# B&R Automation Studio project 8238 (part 23)

#### libTestUse.fun - Exported functions and function blocks
```iecst
(********************************************************************
 * COPYRIGHT -- Herbert Kannegiesser GmbH
 ********************************************************************
 * Library: libTestUse
 * File: libTestUse.fun
 * Author: hunholz
 * Created: March 06, 2012
 ********************************************************************
 * Functions and function blocks of library libTestUse
 ********************************************************************)

FUNCTION_BLOCK TestUser_SetMode (*Versetzt die Anwendung in unterschiedliche Testmodi*)
	VAR_INPUT
		enable : BOOL;
		wMode : UINT;
		pStruc : UDINT;
	END_VAR
	VAR_OUTPUT
		status : UINT;
	END_VAR
	VAR
		_wSetModeState : UINT;
	END_VAR
END_FUNCTION_BLOCK

FUNCTION_BLOCK TestUser_RunTest (*Zyklische Bearbeitung des Tests*)
	VAR_INPUT
		enable : BOOL;
		wMode : UINT;
		pStruc : UDINT;
	END_VAR
	VAR_OUTPUT
		status : UINT;
	END_VAR
	VAR
		_CmdTest : REFERENCE TO TestUser_CmdTest_typ;
		_i : UINT;
		_wCommand : REFERENCE TO UINT;
		_CmdResult : REFERENCE TO ARRAY[0..1] OF UINT;
		_bResult : USINT;
		_wResult : UINT;
		_wXORStatus : UINT;
		_j : UINT;
		_BatchLoad : REFERENCE TO ARRAY[0..3] OF BatchLoad_typ;
		_Batch : REFERENCE TO ARRAY[0..30] OF Batch_typ;
		_BatchUnload : REFERENCE TO ARRAY[0..2] OF Batch_typ;
		_BatchLoadTrig : REFERENCE TO ARRAY[0..3] OF BatchLoadTrig_typ;
		_BatchTrig : REFERENCE TO BatchTrig_typ;
		_BatchUnloadTrig : REFERENCE TO BatchUnloadTrig_typ;
		_xBatchLoadOk : BOOL;
		_xBatchOk : BOOL;
		_xBatchUnloadOk : BOOL;
		_TonShiftClck1 : TON;
		_TonShiftClck2 : TON;
		_wShiftStep : UINT;
		_lBatchNo : UDINT;
		_pBatchNo : REFERENCE TO UDINT;
		_GetTime : DTGetTime;
		_sValue : STRING[10];
		_xBatchForLoadingOk : REFERENCE TO BOOL;
		_enMachineState : REFERENCE TO UDINT;
		_wMachineStateTxt : REFERENCE TO UINT;
		_lMachineStateAtt1 : REFERENCE TO UDINT;
		_lMachineStateAtt2 : REFERENCE TO UDINT;
		_wMachineStateCnt : UINT;
		_Ton1sClck2 : TON;
		_Ton1sClck1 : TON;
	END_VAR
END_FUNCTION_BLOCK

FUNCTION TestUser_StopTask : UINT (*Stoppt Task per Namen*)
	VAR_INPUT
		st_name : UDINT;
	END_VAR
	VAR
		_lTaskIdent : UDINT;
	END_VAR
END_FUNCTION
```

### Program Logical/Standard/Kanlink/KGFrameworkShare/Pkg_mnTestUser/mnTestUser (IEC) - Initialisierung des Test

#### mnTestUserCyclic.st - Cyclic code
```iecst
(********************************************************************
 * COPYRIGHT -- Herbert Kannegiesser GmbH
 ********************************************************************
 * Program: mnTestUser
 * File: mnTestUserCyclic.st
 * Author: hunholz
 * Created: March 07, 2012
 ********************************************************************
 * Implementation of program mnTestUser
 ********************************************************************)

PROGRAM _CYCLIC

(* TODO : Add your code here *)

END_PROGRAM
```

#### mnTestUserInit.st - Initialization code
```iecst
(********************************************************************
 * COPYRIGHT -- Herbert Kannegiesser GmbH
 ********************************************************************
 * Program: mnTestUser
 * File: mnTestUserInit.st
 * Author: hunholz
 * Created: March 07, 2012
 ********************************************************************
 * Implementation of program mnTestUser
 ********************************************************************)

PROGRAM _INIT

	IFmnTest.In.pStrucTest := ADR(_CmdTest);

	_CmdTest.pCmd[1] := ADR(mnMasterCmd.Request.Command);
	_CmdTest.pParamMem[1,1] := ADR(mnMasterCmdAd.SetBatch);
	_CmdTest.pParamSize[1,1] := SIZEOF(mnMasterCmdAd.SetBatch);
	_CmdTest.pCmdResult[1] := ADR(mnMasterCmd.Response);

	_CmdTest.pCmd[2] := ADR(mnLoadCmd.Request.Command);
	_CmdTest.pCmdResult[2] := ADR(mnLoadCmd.Response);

	FOR _i := 0 TO wCountCompMN DO

		_CmdTest.pCmd[3 +_i] := ADR(mnCompCmd[_i].Request.Command);
		_CmdTest.pCmdResult[3 + _i] := ADR(mnCompCmd[_i].Response);

	END_FOR

	_CmdTest.pBatchLoad := ADR(BatchLoad);
	_CmdTest.pBatch := ADR(Batch);
	_CmdTest.pBatchUnload := ADR(BatchUnload);
	_CmdTest.pBatchTrig := ADR(BatchTrig);
	_CmdTest.pBatchLoadTrig := ADR(BatchLoadTrig);
	_CmdTest.pBatchUnloadTrig := ADR(BatchUnloadTrig);

	_CmdTest.pBatchForLoadingOk := ADR(mnMasterStatAd.xBatchTransferDataForLoadingOK);
//
//	_CmdTest.pMachineState := ADR(MachineState.wState);
//	_CmdTest.pMachineStateTxt := ADR(MachineState.wStateTxt);
//	_CmdTest.pMachineStateAtt1 := ADR(MachineState.lStateTxtAtt1);
//	_CmdTest.pMachineStateAtt2 := ADR(MachineState.lStateTxtAtt2);

END_PROGRAM
```

#### mnTestUserExit.st - Exit code
```iecst
(********************************************************************
 * COPYRIGHT -- Herbert Kannegiesser GmbH
 ********************************************************************
 * Program: mnTestUser
 * File: mnTestUserExit.st
 * Author: hunholz
 * Created: March 07, 2012
 ********************************************************************
 * Implementation of program mnTestUser
 ********************************************************************)

PROGRAM _EXIT

(* TODO : Add your code here *)

END_PROGRAM
```

#### mnTestUser.var - Local variables
```iecst
(********************************************************************
 * COPYRIGHT -- Herbert Kannegiesser GmbH
 ********************************************************************
 * Program: mnTestUser
 * File: mnTestUser.var
 * Author: hunholz
 * Created: March 07, 2012
 ********************************************************************
 * Local variables of program mnTestUser
 ********************************************************************)
VAR
	_CmdTest : TestUser_CmdTest_typ;
	_i : UINT;
END_VAR
```

- KanLink Release Notes.docx (binary file, 14716 bytes)
### Package Logical/Standard/Kanlink/CAN - CAN Communication Variables

### CAN.var
```iecst
VAR CONSTANT
	MAX_COMM : USINT := 100;
END_VAR
VAR
	Comm : ARRAY[0..MAX_COMM] OF Comm_typ;
END_VAR
VAR CONSTANT
	COMM_CLEAR : Comm_typ := (0);
END_VAR
```

### CAN.typ
```iecst
TYPE
	WET_CAN : 	STRUCT
		ControlSignals : USINT;
		ControlSignals2 : USINT;
		Category : UINT;
		Customer : UINT;
		Weight : UINT;
	END_STRUCT;
	DRY_CAN : 	STRUCT
		ControlSignals : USINT;
		ControlByte2 : USINT;
		Category : UDINT;
		Weight : UINT;
	END_STRUCT;
	DRY_CAN1 : 	STRUCT
		CustomerCode : UDINT;
		BatchCode : UDINT;
	END_STRUCT;
	DRYCAN_comm_typ : 	STRUCT
		ReadFrame : DRY_CAN;
		WriteFrame : DRY_CAN;
		WriteFrame1 : DRY_CAN1;
		EventRead : BOOL;
		EventWrite : BOOL;
		EventWrite1 : BOOL;
	END_STRUCT;
	Batchpart_typ : 	STRUCT
		Wgt : UINT;
		Customer : UDINT;
	END_STRUCT;
	Comm_typ : 	STRUCT
		BagReady : BOOL;
		Unloading : BOOL;
		DropLoad : BOOL;
		LoadDropped : BOOL;
		Category : UDINT;
		Customer : UDINT;
		BatchID : UDINT;
		Weight : UINT;
		Live : BOOL;
		LiveTime : UINT;
		ReadyToLoad : BOOL;
		Loading : BOOL;
		UnloadFinished : BOOL;
		HaltSys : BOOL;
		Batch_QtyRemaining : UINT;
		LoadRecieved : BOOL;
		Transfer : BOOL;
		Batchpart : ARRAY[0..7]OF Batchpart_typ;
		CategoryStr : STRING[11];
		CustomerStr : STRING[11];
	END_STRUCT;
END_TYPE
```

### Program Logical/Standard/Kanlink/kanlink_map (IEC) - *Custom task to convert Kanlink PLC to eVue Comms

#### Variables.var
```iecst
VAR
	bag_2_wieight : INT;
	doubleDrop : BOOL;
END_VAR
```

#### Cyclic.st
```iecst
PROGRAM _CYCLIC

////SDC1 r43
//Comm[1].Customer	:= wash_com_cust_1;
//Comm[1].Category	:= wash_com_cat_1;
//Comm[1].BatchID		:= DByte_TO_4Byte(ADR(wash_com_batch1_1),ADR(wash_com_batch1_2));
//Comm[1].Weight		:= (wash_com_wt_1 * 10);
//
//Comm[1].BagReady	:= r43.sling_ready;
//r43.open_signal	:= 	Comm[1].DropLoad;
//r43.receive_signal	:= 	Comm[1].LoadDropped;
//IF EDGEPOS(Comm[1].LoadDropped) THEN
//	wash_com_cust_1 := 0;
//	wash_com_cat_1  := 0;
//	wash_com_wt_1  := 0;
//	wash_com_batch1_1 := 0;
//	wash_com_batch1_2 := 0;
//END_IF;
//
////SDC2 r45
//Comm[2].Customer	:= wash_com_cust_2;
//Comm[2].Category	:= wash_com_cat_2;
//Comm[2].BatchID		:= DByte_TO_4Byte(ADR(wash_com_batch1_2),ADR(wash_com_batch2_2));
//Comm[2].Weight		:= (wash_com_wt_2 * 10);
//
//Comm[2].BagReady	:= r45.sling_ready;
//r45.open_signal	:= 	Comm[2].DropLoad;
//r45.receive_signal	:= 	Comm[2].LoadDropped;
//IF EDGEPOS(Comm[2].LoadDropped) THEN
//	wash_com_cust_2 := 0;
//	wash_com_cat_2  := 0;
//	wash_com_wt_2  := 0;
//	wash_com_batch1_2 := 0;
//	wash_com_batch2_2 := 0;
//END_IF;
//
////SDC3 r47
//Comm[3].Customer	:= wash_com_cust_3;
//Comm[3].Category	:= wash_com_cat_3;
//Comm[3].BatchID		:= DByte_TO_4Byte(ADR(wash_com_batch1_3),ADR(wash_com_batch2_3));
//Comm[3].Weight		:= (wash_com_wt_3 * 10);
//
//Comm[3].BagReady	:= r47.sling_ready;
//r47.open_signal	:= 	Comm[3].DropLoad;
//r47.receive_signal	:= 	Comm[3].LoadDropped;
//IF EDGEPOS(Comm[3].LoadDropped) THEN
//	wash_com_cust_3 := 0;
//	wash_com_cat_3  := 0;
//	wash_com_wt_3  := 0;
//	wash_com_batch1_3 := 0;
//	wash_com_batch2_3 := 0;
//END_IF;
//
////CDC8 r110
//Comm[4].Customer	:= wash_com_cust_12;
//Comm[4].Category	:= wash_com_cat_12;
//Comm[4].BatchID		:= DByte_TO_4Byte(ADR(wash_com_batch1_12),ADR(wash_com_batch2_12));
//Comm[4].Weight		:= (wash_com_wt_12 * 10);
//
//Comm[4].BagReady	:= r110.sling_ready;
//r110.open_signal	:= 	Comm[4].DropLoad;
//r110.receive_signal	:= 	Comm[4].LoadDropped;
//IF EDGEPOS(Comm[4].LoadDropped) THEN
//	wash_com_cust_12 := 0;
//	wash_com_cat_12  := 0;
//	wash_com_wt_12  := 0;
//	wash_com_batch1_12 := 0;
//	wash_com_batch2_12 := 0;
//END_IF;
//
////CDC5 r113
//Comm[5].Customer	:= wash_com_cust_13;
//Comm[5].Category	:= wash_com_cat_13;
//Comm[5].BatchID		:= DByte_TO_4Byte(ADR(wash_com_batch1_13),ADR(wash_com_batch2_13));
//Comm[5].Weight		:= (wash_com_wt_13 * 10);
//
//Comm[5].BagReady	:= r113.sling_ready;
//r113.open_signal	:= 	Comm[5].DropLoad;
//r113.receive_signal	:= 	Comm[5].LoadDropped;
//IF EDGEPOS(Comm[5].LoadDropped) THEN
//	wash_com_cust_13 := 0;
//	wash_com_cat_13  := 0;
//	wash_com_wt_13  := 0;
//	wash_com_batch1_13 := 0;
//	wash_com_batch2_13 := 0;
//END_IF;
//
//////CDC6 r68
////Comm[6].Customer	:= wash_com_cust_6;
////Comm[6].Category	:= wash_com_cat_6;
////Comm[6].BatchID		:= DByte_TO_4Byte(ADR(wash_com_batch1_6),ADR(wash_com_batch2_6));
////Comm[6].Weight		:= (wash_com_wt_6 * 10);
////
////Comm[6].BagReady	:= r68.sling_ready;
////r68.open_signal	:= 	Comm[6].DropLoad;
////r68.receive_signal	:= 	Comm[6].LoadDropped;
////IF EDGEPOS(Comm[6].LoadDropped) THEN
////	wash_com_cust_6 := 0;
////	wash_com_cat_6  := 0;
////	wash_com_wt_6  := 0;
////	wash_com_batch1_6 := 0;
////	wash_com_batch2_6 := 0;
////END_IF;
////
//////CDC7 r70
////Comm[7].Customer	:= wash_com_cust_7;
////Comm[7].Category	:= wash_com_cat_7;
////Comm[7].BatchID		:= DByte_TO_4Byte(ADR(wash_com_batch1_7),ADR(wash_com_batch2_7));
////Comm[7].Weight		:= (wash_com_wt_7 * 10);
////
////Comm[7].BagReady	:= r70.sling_ready;
////r70.open_signal	:= 	Comm[7].DropLoad;
////r70.receive_signal	:= 	Comm[7].LoadDropped;
////IF EDGEPOS(Comm[7].LoadDropped) THEN
////	wash_com_cust_7 := 0;
////	wash_com_cat_7  := 0;
////	wash_com_wt_7  := 0;
////	wash_com_batch1_7 := 0;
////	wash_com_batch2_7 := 0;
////END_IF;
////
//////SSL1 r1 - Comm[8]
////
////CSL1 r65
//wash_com_cust_14 	:= UDINT_TO_INT(Comm[14].Customer);
//wash_com_cat_14 		:= UDINT_TO_INT(Comm[14].Category);
//wash_com_wt_14 		:= (Comm[14].Weight/10);
//wash_com_batch1_14	:= Get_Lower2Bytes(Comm[14].BatchID);
//wash_com_batch2_14	:= Get_Higher2Bytes(Comm[14].BatchID);
//
//Comm[14].ReadyToLoad		:= r65.sling_ready;
//r65.xfer_in_progress	:= Comm[14].Unloading;
//
//IF EDGEPOS(r65.fire) THEN
//	wash_com_cust_14 := 0;
//	wash_com_cat_14 := 0;
//	wash_com_wt_14 := 0;
//	wash_com_batch1_14 := 0;
//	wash_com_batch2_14 := 0;
//END_IF;
//
////CSL2 r68
//wash_com_cust_15 	:= UDINT_TO_INT(Comm[15].Customer);
//wash_com_cat_15 	:= UDINT_TO_INT(Comm[15].Category);
//wash_com_wt_15 		:= (Comm[15].Weight/10);
//wash_com_batch1_15	:= Get_Lower2Bytes(Comm[15].BatchID);
//wash_com_batch2_15	:= Get_Higher2Bytes(Comm[15].BatchID);
//
//Comm[15].ReadyToLoad	:= r68.sling_ready;
//r68.xfer_in_progress	:= Comm[15].Unloading;
//
//IF EDGEPOS(r68.fire) THEN
//	wash_com_cust_15 := 0;
//	wash_com_cat_15 := 0;
//	wash_com_wt_15 := 0;
//	wash_com_batch1_15 := 0;
//	wash_com_batch2_15 := 0;
//END_IF;
//
////CSL3 r49
//wash_com_cust_11 	:= UDINT_TO_INT(Comm[11].Customer);
//wash_com_cat_11 	:= UDINT_TO_INT(Comm[11].Category);
//wash_com_wt_11 		:= (Comm[11].Weight/10);
//wash_com_batch1_11	:= Get_Lower2Bytes(Comm[11].BatchID);
//wash_com_batch2_11	:= Get_Higher2Bytes(Comm[11].BatchID);
//
//Comm[11].ReadyToLoad	:= r49.sling_ready;
//r49.xfer_in_progress	:= Comm[11].Unloading;
//
//IF EDGEPOS(r49.fire) THEN
//	wash_com_cust_11 := 0;
//	wash_com_cat_11 := 0;
//	wash_com_wt_11 := 0;
//	wash_com_batch1_11 := 0;
//	wash_com_batch2_11 := 0;
//END_IF;

////CDC2 r70  - DOUBLE DROP>
//Comm[1].Customer	:= wash_com_cust_1;
//Comm[1].Category	:= wash_com_cat_1;
//Comm[1].BatchID		:= DByte_TO_4Byte(ADR(wash_com_batch1_1),ADR(wash_com_batch2_1));
////Comm[1].Weight		:= (wash_com_wt_1 * 10);
//
//bag_4_wieight 		:= WORD_TO_INT(plc_info1);  // 2nd Bag wieght - 1 if the wieght is -0 so we know there is 2 bags.
//doubleDrop			:= (bag_2_wieight > 0);
////Build the batch of 2
//
//IF EDGEPOS(r70.loading_signal) THEN // Decider has ran
//	IF doubleDrop THEN
//		Comm[1].Batch_QtyRemaining := 2;
//	ELSE
//		Comm[1].Batch_QtyRemaining := 1;
//	END_IF;
//END_IF;
//
//IF EDGEPOS(r70.state = 2 ) THEN // Bag arrives in the discharger
//	CASE Comm[1].Batch_QtyRemaining OF
//		1:
//			Comm[1].Batchpart[1].Customer := Comm[1].Customer;
//			Comm[1].Batchpart[1].Wgt := (wash_com_wt_1 * 10);
//			Comm[1].Batchpart[2].Customer := 0;
	//			Comm[1].Batchpart[2].Wgt := 0;
//			Comm[1].Weight := (wash_com_wt_1 *10);
//		2:
//			Comm[1].Batchpart[1].Customer := Comm[1].Customer;
//			Comm[1].Batchpart[1].Wgt := (wash_com_wt_1 * 10);
//			Comm[1].Batchpart[2].Customer := Comm[1].Customer;
//			Comm[1].Batchpart[2].Wgt := (bag_2_wieight * 10);
//			Comm[1].Weight := ((wash_com_wt_1 + bag_2_wieight) *10);
//	END_CASE;
//END_IF;
//
//Comm[1].BagReady	:= r70.sling_ready;
//r70.open_signal	:= 	Comm[1].DropLoad;
//r70.receive_signal	:= 	Comm[1].LoadDropped;
//IF EDGEPOS(Comm[1].LoadDropped) THEN
//	wash_com_cust_1 := 0;
//	wash_com_cat_1  := 0;
//	wash_com_wt_1  := 0;
//	wash_com_batch1_1 := 0;
//	wash_com_batch2_1 := 0;
//	// Count down the loads
//	IF 	Comm[1].Batch_QtyRemaining >= 1 THEN
//		Comm[1].Batch_QtyRemaining := Comm[1].Batch_QtyRemaining - 1;
//	ELSE
//		Comm[1].Batch_QtyRemaining := 0;
//	END_IF;
//END_IF;
//

END_PROGRAM
```

### Package Logical/Robo_Drive_Control - Supertrack Robo Drive Control Package

### Robo_Drive.var - Global variables
```iecst
(********************************************************************
 * COPYRIGHT --
 ********************************************************************
 * Package: FC302
 * File: FC302.var
 * Author: D.Jefferys
 * Created: February 08, 2009
 ********************************************************************
 * Variables of package FC302
 ********************************************************************)
VAR CONSTANT
	AlignReceive : USINT := 1;
	AlignRelease : USINT := 0;
	AlignNone : USINT := 2;
	AlignRest : USINT := 3;
END_VAR
VAR
	StartNode : USINT := 0;
	RB : ARRAY[0..MaxRobo] OF FC302_Drive_Typ := [8(0)];
END_VAR
VAR RETAIN
	RB_Retain : ARRAY[0..MaxRobo] OF FC302_Drive_Retain_Typ;
	RB_Posn : ARRAY[0..MaxRobo] OF FC302_Position_Type;
	RB_Perm : ARRAY[0..MaxRobo] OF FC302_Drive_Permanent_Typ;
END_VAR
VAR
	RB_PosnName : ARRAY[0..MaxRobo] OF RoboPositionNames;
	MonitorIdx : USINT := 0;
END_VAR
```

### Library Logical/Robo_Drive_Control/FC302 (IEC) - FC302 Functions Library

#### FC302.typ - Exported data types
```iecst
(********************************************************************
 * COPYRIGHT --
 ********************************************************************
 * Library: FC302
 * File: FC302.typ
 * Author: D.Jefferys
 * Created: February 12, 2009
 ********************************************************************
 * Data types of library FC302
 ********************************************************************)

TYPE
	RoboPositionNames : 	STRUCT
		Name : ARRAY[0..MaxPositions]OF UINT;
		Extra : ARRAY[0..MaxPositions]OF UINT;
	END_STRUCT;
	FC302_Position_Type : 	STRUCT
		Lift : FC032_Drive_Positions_Type;
		Rotate : FC032_Drive_Positions_Type;
	END_STRUCT;
	FC032_Drive_Positions_Type : 	STRUCT
		RefOffset : DINT;
		MaxSpeed : DINT; (*Max speed in mm/sec*)
		CycleCount : DINT; (*Read only for TrackView display only*)
		PositionNow : DINT;
		OperationMode : DINT; (*0=Normal Sequence 1=Manual Operation*)
		IOStatus : DINT; (*I/O Transmitted to TrackView*)
		Monitor : DINT; (*Monitor Values*)
		SeqStep : DINT; (*Sequence Step*)
		Posn : ARRAY[0..MaxPositions]OF DINT;
	END_STRUCT;
	FC302_Drive_Permanent_Typ : 	STRUCT
		Lift : FC302_LiftPermenant;
		Rotate : FC302_RotatePermenant;
	END_STRUCT;
	FC302_LiftPermenant : 	STRUCT
		CycleCount : DINT;
	END_STRUCT;
	FC302_RotatePermenant : 	STRUCT
		CycleCount : DINT;
	END_STRUCT;
	FC302_Drive_Retain_Typ : 	STRUCT
		Lift : FC302_LiftRemanent;
		Rotate : FC302_RotateRemanent;
	END_STRUCT;
	FC302_Drive_Typ : 	STRUCT
		Lift : FC302_Lift;
		Rotate : FC302_Rotate;
	END_STRUCT;
	FC302_RotateRemanent : 	STRUCT
		PosnRef : DINT;
	END_STRUCT;
	FC302_LiftRemanent : 	STRUCT
		PosnRef : DINT;
	END_STRUCT;
	FC302_Lift : 	STRUCT
		SeqStep : UINT;
		Encoder : DINT; (*Encoder raw value from card*)
		PosnActRaw : UDINT; (*Encoder position actual value always positive*)
		PosnAct : DINT;
		PosnNow : DINT; (*Actual calculated position in 100th of mm*)
		PulsePer10th_mm : REAL;
		DistRemain : DINT;
		mmPerHz : REAL;
		RunHz : UINT; (*Calculated run frequency *)
		StopDist : DINT;
		RunForwards : BOOL;
		RunReverse : BOOL;
		RunFreq : UINT; (*Actual drive running frequency *)
		RampStart : DINT; (*Final Ramp Start (ms)*)
		RampTime : DINT; (*Final Ramp Time (ms)*)
		RampMax : DINT; (*Final Ramp Max Time (ms)*)
		CAN : FC302_CAN_Typ;
		Scan : FC302_CAN_Scan_Typ;
		CTW : FC302_CTW_Typ;
		STW : FC302_STW_Typ;
		SeqIn : FC302_ControlIn; (*Inputs from PLC Sequence*)
		SeqOut : FC302_ControlOut; (*Outputs to PLC Sequence*)
		ParaList : ARRAY[0..59]OF FC302_Parameter_Typ;
		Motor : FC302_Motor_Info;
		ParamWrite : FC302_ParamWrite;
		ParameterCount : UINT;
		ModuleOK : BOOL;
	END_STRUCT;
	FC302_Rotate : 	STRUCT
		SeqStep : UINT;
		Encoder : DINT; (*Encoder raw value from card*)
		PosnActRaw : UDINT; (*Encoder position actual value always positive*)
		PosnAct : DINT;
		PosnNow : DINT; (*Actual calculated position in 100ths of degrees*)
		PulsePer100th_Deg : REAL;
		DistRemain : DINT;
		mmPerHz : REAL;
		RunHz : UINT; (*Calculated run frequency *)
		StopDist : DINT;
		RefOffsetDeg : UINT; (*Degrees from 0 of the reference proximity switch in 100ths 50 = 5000*)
		RunForwards : BOOL;
		RunReverse : BOOL;
		RunFreq : UINT; (*Actual drive running frequency *)
		RampStart : DINT; (*Final Ramp Start (ms)*)
		RampTime : DINT; (*Final Ramp Time (ms)*)
		RampMax : DINT; (*Final Ramp Max Time (ms)*)
		CAN : FC302_CAN_Typ;
		CTW : FC302_CTW_Typ;
		STW : FC302_STW_Typ;
		Scan : FC302_CAN_Scan_Typ;
		SeqIn : FC302_ControlIn; (*Inputs from PLC Sequence*)
		SeqOut : FC302_ControlOut; (*Outputs to PLC Sequence*)
		ParaList : ARRAY[0..59]OF FC302_Parameter_Typ;
		Motor : FC302_Motor_Info;
		ParamWrite : FC302_ParamWrite;
		ParameterCount : UINT;
		ModuleOK : BOOL;
	END_STRUCT;
	FC302_ControlIn : 	STRUCT
		DoRef : BOOL;
		AutoTunePosn : UINT; (*Auto tune position number*)
		AutoTuneReceive : BOOL; (*Auto tune for receive alignment*)
		sDevice : STRING[10]; (*CAN Device eg. "SS1.IF2"*)
		sParTblName : STRING[10]; (*Taskname of parameter table*)
		Node : USINT; (*CAN Node of drive*)
		DisableDrive : BOOL; (*Input - Enable drive to run the motor*)
		I_RefPosn : BOOL; (*Input - PLC Input for reference position*)
		I_ForwardLimitOk : BOOL; (*Input - PLC Input for Top/Clockwise limit *)
		I_ReverseLimitOk : BOOL; (*Input - PLC Input for Bottom/Anti-clockwise limit*)
		I_RailOkRelease : BOOL; (*Input - PLC Input for Rail aligned for bag to leave*)
		I_RailOkReceive : BOOL; (*Input - PLC Input for Rail aligned to Receive a bag*)
		JogForwards : BOOL;
		JogReverse : BOOL;
		EStop : BOOL; (*Input - System emergency stop - will stop drive*)
		PosnReq : DINT; (*Input - Required position in mm 10ths / 100ths Deg *)
		MaxSpeed : DINT; (*Input - Max running speed mm/sec *)
		PowerSave : BOOL; (*Input - Not Busy so save power move slower*)
		RailAlign : USINT; (*Input - Rail Align Requirement*)
		Run : BOOL; (*Input - Run Drive*)
	END_STRUCT;
	FC302_ControlOut : 	STRUCT
		PosnNow : INT; (*Output - Actual Position in mm*)
		PosnOk : BOOL; (*Output - Current position ok for release*)
		DriveDisabled : BOOL; (*Output - Drive acknoledge Enable Movement is off*)
		RefComplete : BOOL; (*Output - Drive is referenced and ready to run*)
		AutoTunePosn : UINT; (*Auto tune position number*)
		Status : UINT; (*Output - Drive sequence status 0 = all ok ready*)
	END_STRUCT;
	FC302_CAN_Scan_Typ : 	STRUCT
		Start : TIME;
		End : TIME;
		LastScan : UINT;
		MinScan : UINT;
		MaxScan : UINT;
		StartTrig : BOOL;
		EndTrig : BOOL;
	END_STRUCT;
	FC302_CAN_Typ : 	STRUCT
		ModuleOk : BOOL; (*Module OK*)
		NodeStatus : UINT; (*Node Status*)
		ControlWord : UINT; (*Control Word*)
		StatusWord : UINT; (*Status Word*)
		TargetVelocity : UINT; (*Target Velocity*)
		ControlEffort : UINT; (*Control Effort*)
	END_STRUCT;
	FC302_Parameter_Typ : 	STRUCT
		index : UINT;
		subindex : USINT;
		datalen : USINT;
		data : UDINT;
	END_STRUCT;
	FC302_ParamWrite : 	STRUCT
		ErrorCount : UINT;
		Index : UINT;
		SubIndex : USINT;
	END_STRUCT;
	FC302_STW_Typ : 	STRUCT  (*Status Word Type*)
		ControlReady : BOOL; (*0 = Off tripped  1 = Controls ready*)
		DriveReady : BOOL; (*0 = Drive not ready 1 = Drive ready*)
		CoastingStop : BOOL; (*0 = Drive has released the motor 1 = Operation enabled*)
		Trip : BOOL; (*0 = No error 1 = Drive Tripped*)
		Error : BOOL; (*0 = No error 1 = Drive has an error but not tripped*)
		NotUsed : BOOL;
		TripLock : BOOL; (*0 = No error 1 = Drive is tripped and locked*)
		Warning : BOOL; (*0 = No error 1 = Drive warning has occured*)
		SpeedReference : BOOL; (*0 = Speed not equal to reference 1 = Speed equals reference*)
		BusOperation : BOOL; (*0 = Local operation no bus control 1 = Bus operation enabled *)
		FreqLimitOk : BOOL; (*0 = Frequency limit reached high or low 1 = Between the limits*)
		DriveOverTemp : BOOL; (*0 = Temperature ok 1 = Drive stopped because of over temperature will resume *)
		DriveVoltageFault : BOOL; (*0 = Voltage ok 1 = Drive DC voltage too high or low*)
		DriveTorqueLimit : BOOL; (*0 = Torque ok 1 = Torque (Current) limit in param 4-18 has been exceded *)
		ThermalTimerLimit : BOOL; (*0 = Timer ok 1 = One of the thermal protection timers has exceeded 100%*)
		InOperation : BOOL; (*0 = Stopped 1 = Drive running greater then 0 Hz*)
	END_STRUCT;
	FC302_Motor_Info : 	STRUCT  (*Current Motor Information *)
		Value : INT;
	END_STRUCT;
	FC302_CTW_Typ : 	STRUCT  (*Control Word Type*)
		ExtRefSelectionLSB : BOOL; (*Used to select between the 4 reference values in parameter 3-10*)
		ExtRefSelectionMSB : BOOL; (*Used to select between the 4 reference values in parameter 3-10*)
		DC_Brake : BOOL; (*0 = DC Brake 1 = Ramp *)
		Coasting : BOOL; (*0 = Coasting 1 = No Coasting, selecting 0 will shut off the output transistors.*)
		QuickStop : BOOL; (*0 = QuickStop 1= Ramp, selecting 0 will use parameter 3-81 quick stop ramp time.*)
		HoldOutputFreq : BOOL; (*0 = Hold 1= Ramp, always use Ramp*)
		RampStopStart : BOOL; (*0 = Ramp stop 1 = Start, Normal stsrt / stop*)
		ResetTrip : BOOL; (*0 = Nothing 1 = Reset Trip*)
		Jog : BOOL; (*0 = Normal 1 = Jog, Jog frequency set by parameter 3-19*)
		RampSelection : BOOL; (*0 = Ramp 1 1 = Ramp 2, Select between ramp 1 and 2 3-40 to 3-47 or 3-50 to 3-57*)
		DataValid : BOOL; (*0 = Not Valid 1 = Data Valid, If not valid then the whole control word is ignored.*)
		Relay01Active : BOOL; (*0 = No function*)
		Relay02Active : BOOL; (*0 = No function*)
		ParaSetUpLSB : BOOL; (*Used to select between the 4 different parameter setups*)
		ParaSetUpMSB : BOOL; (*Used to select between the 4 different parameter setups*)
		Reverse : BOOL; (*0 = No reversing 1 = Reversing*)
	END_STRUCT;
END_TYPE
```

#### FC302.var - Exported constants
```iecst
(********************************************************************
 * COPYRIGHT --
 ********************************************************************
 * Library: FC302
 * File: FC302.var
 * Author: D.Jefferys
 * Created: February 12, 2009
 ********************************************************************
 * Constants of library FC302
 ********************************************************************)
VAR CONSTANT
	posnNameNone : UINT := 0;
	posnNameTop : UINT := 1;
	posnNameTopBagIn : UINT := 2;
	posnNameTopBagOut : UINT := 3;
	posnNameBottom : UINT := 4;
	posnNameBottomBagIn : UINT := 5;
	posnNameBottomBagOut : UINT := 6;
	posnNameMiddle : UINT := 7;
	posnNameMiddleBagIn : UINT := 8;
	posnNameMiddleBagOut : UINT := 9;
	posnNameHighLevel : UINT := 10;
	posnNameHighLevelBagIn : UINT := 11;
	posnNameHighLevelBagOut : UINT := 12;
	posnNameLowLevel : UINT := 13;
	posnNameLowLevelBagIn : UINT := 14;
	posnNameLowLevelBagOut : UINT := 15;
	posnNameMidLevel : UINT := 16;
	posnNameMidLevelBagIn : UINT := 17;
	posnNameMidLevelBagOut : UINT := 18;
	posnNameDocking : UINT := 19;
	posnNameDummy : UINT := 20;
	posnNameLoading : UINT := 21;
	posnNameLine : UINT := 22;
	posnNameParking : UINT := 23;
	posnNameRecirculation : UINT := 24;
	posnNameSafety : UINT := 25;
	posnNameWeighing : UINT := 26;
	posnExtraNone : UINT := 0;
	posnExtraLine1 : UINT := 1;
	posnExtraLine2 : UINT := 2;
	posnExtraLine3 : UINT := 3;
	posnExtraLine4 : UINT := 4;
	posnExtraLine5 : UINT := 5;
	posnExtraLine6 : UINT := 6;
	posnExtraLine7 : UINT := 7;
	posnExtraLine8 : UINT := 8;
	posnExtraLine9 : UINT := 9;
	posnExtraLine10 : UINT := 10;
	posnExtraLine11 : UINT := 11;
	posnExtraLine12 : UINT := 12;
	posnExtraLine13 : UINT := 13;
	posnExtraLine14 : UINT := 14;
	posnExtraLine15 : UINT := 15;
	posnExtraLine16 : UINT := 16;
	posnExtraLine17 : UINT := 17;
	posnExtraLine18 : UINT := 18;
	posnExtraLine19 : UINT := 19;
	posnExtraLine20 : UINT := 20;
	posnExtraLine21 : UINT := 21;
	posnExtraLine22 : UINT := 22;
	posnExtraLine23 : UINT := 23;
	posnExtraLine24 : UINT := 24;
	posnExtraLine25 : UINT := 25;
	posnExtraLine26 : UINT := 26;
	posnExtraLine27 : UINT := 27;
	posnExtraLine28 : UINT := 28;
	posnExtraLine29 : UINT := 29;
	posnExtraSeqHeader1 : UINT := 101;
	posnExtraSeqHeader2 : UINT := 102;
	posnExtraSeqHeader3 : UINT := 103;
	posnExtraSeqHeader4 : UINT := 104;
	posnExtraSeqHeader5 : UINT := 105;
	posnExtraSeqHeader6 : UINT := 106;
	posnExtraSeqHeader7 : UINT := 107;
	posnExtraSeqHeader8 : UINT := 108;
	posnExtraSeqHeader9 : UINT := 109;
	posnExtraSeqHeader10 : UINT := 110;
	posnExtraSeqHeader11 : UINT := 111;
	posnExtraSeqHeader12 : UINT := 112;
	posnExtraSeqHeader13 : UINT := 113;
	posnExtraSeqHeader14 : UINT := 114;
	posnExtraSeqHeader15 : UINT := 115;
	posnExtraSeqHeader16 : UINT := 116;
	posnExtraSeqHeader17 : UINT := 117;
	posnExtraSeqHeader18 : UINT := 118;
	posnExtraSeqHeader19 : UINT := 119;
	posnExtraSeqHeader20 : UINT := 120;
	posnExtraSeqHeader21 : UINT := 121;
	posnExtraSeqHeader22 : UINT := 122;
	posnExtraSeqHeader23 : UINT := 123;
	posnExtraSeqHeader24 : UINT := 124;
	posnExtraSeqHeader25 : UINT := 125;
	posnExtraSeqHeader26 : UINT := 126;
	posnExtraSeqHeader27 : UINT := 127;
	posnExtraSeqHeader28 : UINT := 128;
	posnExtraSeqHeader29 : UINT := 129;
	posnExtraSeqHeader30 : UINT := 130;
	posnExtraSeqHeader31 : UINT := 131;
	posnExtraSeqHeader32 : UINT := 132;
	posnExtraSeqHeader33 : UINT := 133;
	posnExtraSeqHeader34 : UINT := 134;
	posnExtraSeqHeader35 : UINT := 135;
	posnExtraSeqHeader36 : UINT := 136;
	posnExtraSeqHeader37 : UINT := 137;
	posnExtraSeqHeader38 : UINT := 138;
	posnExtraSeqHeader39 : UINT := 139;
	posnExtraSeqHeader40 : UINT := 140;
	posnExtraSeqHeader41 : UINT := 141;
	posnExtraSeqHeader42 : UINT := 142;
	posnExtraSeqHeader43 : UINT := 143;
	posnExtraSeqHeader44 : UINT := 144;
	posnExtraSeqHeader45 : UINT := 145;
	posnExtraSeqHeader46 : UINT := 146;
	posnExtraSeqHeader47 : UINT := 147;
	posnExtraSeqHeader48 : UINT := 148;
	posnExtraSeqHeader49 : UINT := 149;
	MaxRobo : USINT := 7;
	MaxPositions : USINT := 29;
	ModeNothing : UINT := 0;
	ModeReference : UINT := 1;
	ModeManualMove : UINT := 2;
	ModePosnTune : UINT := 3;
	ModeMovePosn : UINT := 4;
	ActionNothing : UINT := 0;
	ActionMoveUp : UINT := 1;
	ActionMoveDown : UINT := 2;
	ActionMoveLeft : UINT := 3;
	ActionMoveRight : UINT := 4;
	FC302_SEQ_OK : USINT := 0;
	FC302_SEQ_Disabled : USINT := 1;
	FC302_SEQ_IndexError : USINT := 2;
	FC302_SEQ_SetCANPreOperational : USINT := 3;
	FC302_SEQ_RestartCANnode : USINT := 4;
	FC302_SEQ_ReadParameterTable : USINT := 5;
	FC302_SEQ_WriteParameters : USINT := 6;
	FC302_SEQ_StoreParameters : USINT := 7;
	FC302_SEQ_CheckParamStored : USINT := 8;
	FC302_SEQ_StartCANnode : USINT := 9;
	FC302_SEQ_WaitDriveOperational : USINT := 10;
	FC302_SEQ_Referencing : USINT := 11;
	FC302_SEQ_MotorWiringFault : USINT := 12;
	FC302_SEQ_RefNotFound : USINT := 13;
	FC302_SEQ_ParameterError : USINT := 14;
	FC302_SEQ_RefSwitchFault : USINT := 15;
	FC302_SEQ_AutoTune : USINT := 16;
	FC302_SEQ_Jog : USINT := 17;
	FC302_SEQ_ReleaseSwitchFault : USINT := 18;
	FC302_SEQ_ReceiveSwitchFault : USINT := 19;
	FC302_SEQ_RailNotAligned : USINT := 20;
	FC302_STW_Trip : USINT := 101;
	FC302_STW_Error : USINT := 102;
	FC302_STW_TripLock : USINT := 103;
	FC302_STW_Warning : USINT := 104;
	FC302_STW_DriveOverTemp : USINT := 105;
	FC302_STW_DriveVoltageFault : USINT := 106;
	FC302_STW_DriveTorqueLimit : USINT := 107;
	FC302_STW_ThermalTimeLimit : USINT := 108;
END_VAR
```

#### FC302.fun - Exported functions and function blocks
```iecst
(********************************************************************
 * COPYRIGHT --
 ********************************************************************
 * Library: FC302
 * File: FC302.fun
 * Author: D.Jefferys
 * Created: February 12, 2009
 ********************************************************************
 * Functions and function blocks of library FC302
 ********************************************************************)

FUNCTION_BLOCK FC302_WriteParam
	VAR_INPUT
		enable : BOOL;
		pDevice : UDINT; (*Add your parameter comment*)
		node : USINT; (*Add your parameter comment*)
		index : UINT; (*Add your parameter comment*)
		subindex : USINT; (*Add your parameter comment*)
		data : UDINT; (*Add your parameter comment*)
		bytelen : USINT; (*Add your parameter comment*)
	END_VAR
	VAR_OUTPUT
		status : UINT; (*Add your parameter comment*)
	END_VAR
	VAR
		CANopenSDOWrite8_0 : CANopenSDOWrite8;
	END_VAR
END_FUNCTION_BLOCK

FUNCTION_BLOCK FC302_ReadSTW (*FC302 Read Status Word*)
	VAR_INPUT
		StatusWord : UINT; (*Add your parameter comment*)
	END_VAR
	VAR_OUTPUT
		STW : FC302_STW_Typ; (*Add your parameter comment*)
	END_VAR
END_FUNCTION_BLOCK

FUNCTION_BLOCK FC302_WriteCTW (*Control Word build*)
	VAR_INPUT
		CTW : FC302_CTW_Typ; (*Add your parameter comment*)
	END_VAR
	VAR_OUTPUT
		ControlWord : UINT; (*Add your parameter comment*)
	END_VAR
	VAR
		LocalControlWord : UINT;
	END_VAR
END_FUNCTION_BLOCK

FUNCTION_BLOCK FC302_ReadParamTbl
	VAR_INPUT
		Enable : BOOL;
		adrTableName : UDINT;
		adrDestTable : UDINT;
		ParamLimit : UINT;
	END_VAR
	VAR_OUTPUT
		ParamCount : UINT;
		Status : UINT;
	END_VAR
	VAR
		DatObjInfo_0 : DatObjInfo;
		DatObjRead_0 : DatObjRead;
	END_VAR
END_FUNCTION_BLOCK

FUNCTION_BLOCK FC302_ReadParam (*Read Parameter from Danfoss FC302*)
	VAR_INPUT
		enable : BOOL; (*Add your parameter comment*)
		pDevice : UDINT; (*Add your parameter comment*)
		node : USINT; (*Add your parameter comment*)
		index : UINT; (*Add your parameter comment*)
		subindex : USINT; (*Add your parameter comment*)
	END_VAR
	VAR_OUTPUT
		data : UDINT; (*Add your parameter comment*)
		status : UINT; (*Add your parameter comment*)
	END_VAR
	VAR
		bytelen : USINT; (*Add your parameter comment*)
		CANopenSDORead8_0 : CANopenSDORead8;
	END_VAR
END_FUNCTION_BLOCK
```

#### FC302_WriteParam.ab - Write Parameter to Danfoss FU302 Drive
```automation-basic
(********************************************************************
 * COPYRIGHT --
 ********************************************************************
 * Program: CAN_Open
 * File: FU302_WriteParam.ab
 * Author: D.Jefferys
 * Created: February 10, 2009
 ********************************************************************
 * Implementation of program CAN_Open
 ********************************************************************)

(*TODO: Add your comment here*)
FUNCTION_BLOCK FC302_WriteParam

	CANopenSDOWrite8_0.enable 	= enable
	CANopenSDOWrite8_0.pDevice 	= pDevice
	CANopenSDOWrite8_0.node 	= node
	CANopenSDOWrite8_0.index 	= $2000 + index
	CANopenSDOWrite8_0.subindex = subindex
	memset(ADR(CANopenSDOWrite8_0.data0),0,8)
	memcpy(ADR(CANopenSDOWrite8_0.data0),ADR(data),4)
	CANopenSDOWrite8_0.datalen 	= bytelen

	CANopenSDOWrite8_0 FUB CANopenSDOWrite8()

	status = CANopenSDOWrite8_0.status

END_FUNCTION_BLOCK
```

#### FC302_ReadSTW.ab - FC302 Read Status Word
```automation-basic
(********************************************************************
 * COPYRIGHT --
 ********************************************************************
 * Program: CAN_Open
 * File: FC302_ReadSTW.ab
 * Author: D.Jefferys
 * Created: February 11, 2009
 ********************************************************************
 * Implementation of program CAN_Open
 ********************************************************************)

(*FC302 Read Status Word*)
FUNCTION_BLOCK FC302_ReadSTW

	STW.ControlReady   		= BIT_TST(StatusWord,0)
	STW.DriveReady			= BIT_TST(StatusWord,1)
	STW.CoastingStop		= BIT_TST(StatusWord,2)
	STW.Trip				= BIT_TST(StatusWord,3)
	STW.Error				= BIT_TST(StatusWord,4)
	STW.NotUsed				= BIT_TST(StatusWord,5)
	STW.TripLock			= BIT_TST(StatusWord,6)
	STW.Warning				= BIT_TST(StatusWord,7)
	STW.SpeedReference		= BIT_TST(StatusWord,8)
	STW.BusOperation		= BIT_TST(StatusWord,9)
	STW.FreqLimitOk			= BIT_TST(StatusWord,10)
	STW.InOperation			= BIT_TST(StatusWord,11)
	STW.DriveOverTemp		= BIT_TST(StatusWord,12)
	STW.DriveVoltageFault	= BIT_TST(StatusWord,13)
	STW.DriveTorqueLimit	= BIT_TST(StatusWord,14)
	STW.ThermalTimerLimit	= BIT_TST(StatusWord,15)

END_FUNCTION_BLOCK
```

#### FC302_WriteCTW.ab - FC302 Write Control Word
```automation-basic
(********************************************************************
 * COPYRIGHT --
 ********************************************************************
 * Library: FC302
 * File: FC302_WriteCTW.ab
 * Author: D.Jefferys
 * Created: February 12, 2009
 ********************************************************************
 * Implementation of library FC302
 ********************************************************************)

(*Control Word build*)
FUNCTION_BLOCK FC302_WriteCTW

	LocalControlWord = 0

	IF CTW.ExtRefSelectionLSB THEN
		LocalControlWord = LocalControlWord + 1
	ENDIF
	IF CTW.ExtRefSelectionMSB THEN
		LocalControlWord = LocalControlWord + 2
	ENDIF
	IF CTW.DC_Brake THEN
		LocalControlWord = LocalControlWord + 4
	ENDIF
	IF CTW.Coasting THEN
		LocalControlWord = LocalControlWord + 8
	ENDIF
	IF CTW.QuickStop THEN
		LocalControlWord = LocalControlWord + 16
	ENDIF
	IF CTW.HoldOutputFreq THEN
		LocalControlWord = LocalControlWord + 32
	ENDIF
	IF CTW.RampStopStart THEN
		LocalControlWord = LocalControlWord + 64
	ENDIF
	IF CTW.ResetTrip THEN
		LocalControlWord = LocalControlWord + 128
	ENDIF
	IF CTW.Jog THEN
		LocalControlWord = LocalControlWord + 256
	ENDIF
	IF CTW.RampSelection THEN
		LocalControlWord = LocalControlWord + 512
	ENDIF
	IF CTW.DataValid THEN
		LocalControlWord = LocalControlWord + 1024
	ENDIF
	IF CTW.Relay01Active THEN
		LocalControlWord = LocalControlWord + 2048
	ENDIF
	IF CTW.Relay02Active THEN
		LocalControlWord = LocalControlWord + 4096
	ENDIF
	IF CTW.ParaSetUpLSB THEN
		LocalControlWord = LocalControlWord + 8192
	ENDIF
	IF CTW.ParaSetUpMSB THEN
		LocalControlWord = LocalControlWord + 16384
	ENDIF
	IF CTW.Reverse THEN
		LocalControlWord = LocalControlWord + 32768
	ENDIF

	ControlWord = LocalControlWord

END_FUNCTION_BLOCK
```

#### FC302_ReadParamTbl.ab - Read from a parameter table
```automation-basic
(********************************************************************
 * COPYRIGHT --
 ********************************************************************
 * Library: FC302
 * File: ReadParamTbl.ab
 * Author: D.Jefferys
 * Created: February 13, 2009
 ********************************************************************
 * Implementation of library FC302
 ********************************************************************)

(*Read from a parameter table*)
FUNCTION_BLOCK FC302_ReadParamTbl

	IF Enable THEN

		Status 		= $FFFF ;Set to busy
		ParamCount 	= 0

		DatObjInfo_0.enable = TRUE
		DatObjInfo_0.pName = adrTableName
		DatObjInfo_0 FUB DatObjInfo()

		IF (DatObjInfo_0.status = 0) THEN

			ParamCount 	= UINT(DatObjInfo_0.len / 8)

			IF (ParamCount <= ParamLimit) THEN

				DatObjRead_0.enable 		= TRUE
				DatObjRead_0.ident 			= DatObjInfo_0.ident
				DatObjRead_0.Offset 		= 0
				DatObjRead_0.pDestination 	= adrDestTable
				DatObjRead_0.len 			= DatObjInfo_0.len
				DatObjRead_0 FUB DatObjRead()

				IF DatObjRead_0.status = 0 THEN
					Status = 0 ;Set status to finished
				ENDIF

			ELSE
				Status = 1 ;Too may parameters
			ENDIF

		ENDIF

	ENDIF

END_FUNCTION_BLOCK
```

#### FC302_ReadParam.ab - Read Parameter from Danfoss FC302
```automation-basic
(********************************************************************
 * COPYRIGHT --
 ********************************************************************
 * Library: FC302
 * File: FC302_ReadParam.ab
 * Author: D.Jefferys
 * Created: February 13, 2009
 ********************************************************************
 * Implementation of library FC302
 ********************************************************************)

(*Read Parameter from Danfoss FC302*)
FUNCTION_BLOCK FC302_ReadParam

	status = 65535 ;Busy

	CANopenSDORead8_0.enable 	= enable
	CANopenSDORead8_0.pDevice 	= pDevice
	CANopenSDORead8_0.node 		= node
	CANopenSDORead8_0.index 	= $2000 + index
	CANopenSDORead8_0.subindex 	= subindex

	CANopenSDORead8_0 FUB CANopenSDORead8()

	IF (CANopenSDORead8_0.status = 0) THEN
		data = 0
		memcpy(ADR(data),ADR(CANopenSDORead8_0.data0),CANopenSDORead8_0.datalen)
		status = CANopenSDORead8_0.status
	ENDIF

END_FUNCTION_BLOCK
```

### Data object Logical/Robo_Drive_Control/Param_3kw (Simple, version 4.00.0) - Parameters 3kW Star from Expo

#### Param_3kw.dat
```
(********************************************************************
 * COPYRIGHT --
 ********************************************************************
 * Data object: Param_2kwStar
 * File: Param_2kwStar.dat
 * Author:  D.Jefferys
 * Created: February 12, 2009
 ********************************************************************
 * Data object file: Param_2kwStar.dat
 ********************************************************************)

;Version 4.01 18/12/2012 T.R. Created 3kw instance based on 2.2kw version 4.00
;CAN Module Switch Settings
;--------------------------

;Baudrate
;8 on  7 on  Par 10-01
;8 on  7 off 500kbps
;8 off 7 on  250kbps
;8 off 7 off 125kbps

;Node Number Binary
;1 = 1s
;2 = 2s
;3 = 4s
;4 = 8s
;5 = 16s
;6 = 32s

;
;	!!! DO NOT CHANGE THE SEQUENCE OF THE PARAMETERS
;
; FU parameter to the Ubertragung (only parameter, which deviates from the default values)
;
; 3 kW Star
;
; Index, Subindex, Datatype (Bytes), Setting (DINT) ; Comments
0002,00,01,00000001	; [000] 00-02, Motor Speed 0 - RPM, 1 - Hz
0001,00,01,00000000	; [001] 00-01, Language 0 - English, 1 - German
0011,00,01,00000001	; [002] 00-11, Edit Setup 1
0190,00,01,00000002	; [003] 01-90, Motor Thermal Protection, 2 - Thermistor
0040,00,01,00000000 ; [004] 00-40, Hand On Key on LCP 0 - Disabled No Function
0381,00,04,00000020 ; [005] 03-81, QuickStop ramp time 100 - 1s
0458,00,01,00000001	; [006] 04-58, Missing motor phase function, 1 - Trip 100ms
0854,00,01,00000001	; [007] 08-54, Reversing select 1 - Bus only 3 - Bus and Terminal
0211,00,02,00000300	; [008] 02-11, Brake resistor 100 Ohm
0212,00,04,00001500	; [009] 02-12, Brake power limit 200 Watt
0213,00,01,00000002	; [010] 02-13, Brake check 2 - Alarm
1426,00,01,00000000 ; [011] 14-26, Trip delay at inverter fault 0 = Disabled
0803,00,04,00000002 ; [012] 08-03, Control Word Timeout Time 10 = 1Sec
0804,00,01,00000002	; [013] 08-04, Control Word Timeout Function 2 - Stop with auto restart
0801,00,01,00000000	; [014] 08-01, Control Site, 0 - Controlword & digital only
0223,00,01,00000005	; [015] 02-23, Active brake delay 0,3 s
1761,00,01,00000002	; [016] 17-61, Encoder Signal Monitoring (Encoder faulty), 2 - Trip
1710,00,01,00000001	; [017] 17-10, Encoder Signal Type 1 - TTL
1711,00,02,00001024	; [018] 17-11, Encoder Resolution 1024 Pulse
0430,00,01,00000001 ; [019] 04-30, Motor Feedback Loss Function, 1 - Warning, 2* - Trip
0431,00,02,00000300 ; [020] 04-31, Motor Feedback Speed Error RPM, 0-600, 300*
0226,00,02,00005000	; [021] 02-26, Torque Ref, 50,00%
0228,00,02,00000200	; [022] 02-28, Gain Boost Factor, 2,00% 0-4% ***************************
0519,00,01,00000003	; [023] 05-19, Terminal 37 Safe Stop, 3 - Safe Stop Warning
0120,00,04,00000300	; [024] 01-20, Motor Power 3kW
0101,00,01,00000003	; [025] 01-01, Motor Control Principle, 3 - Flux with motor feedback
0122,00,02,00000400	; [026] 01-22, Motor voltage 400 V
0123,00,02,00000050	; [027] 01-23, Motor frequency 50 Hz
0162,00,02,00000100	; [028] 01-62, Slip compenstation 100%
0410,00,01,00000002	; [029] 04-10, Motor speed direction, 2 - both directions
0540,00,01,00000032	; [030] 05-40, [0] Relay 1 Function, 32 - Mech brake ctrl
0540,01,01,00000032	; [031] 05-40, [1] Relay 2 Function, 32 - Mech brake ctrl
0802,00,01,00000003 ; [032] 08-02, Control Site 3 - Option A CAN Bus
0102,00,01,00000002	; [033] 01-02, Flux Motor Feeback Source 2 - MCB102
0125,00,02,00001420	; [034] 01-25, Motor nominal speed 1420 rpm
0702,00,02,00000070	; [035] 07-02, Speed PID proportionl gain 0,070
0700,00,01,00000002	; [036] 07-00, Speed PID Feedback Source 2 - MCB102
0172,00,01,00000006	; [037] 01-72, Start function, 6 - Hoist Mech. Brake Rel
0210,00,01,00000001	; [038] 02-10, Brake Function, 1 - Resistor brake
1410,00,01,00000005	; [039] 14-10, Mains failure, 3 - Coasting 5 - Kenetic backup , trip
0193,00,01,00000006	; [040] 01-93, Thermistor source, 6 - Digital Input 33
0100,00,01,00000001	; [041] 01-00, Configuration mode, 1 - Closed loop with encoder
0139,00,01,00000004	; [042] 01-39, Motor poles, 4
0511,00,01,00000000	; [043] 05-11, Terminal 19, 0 - No Operation
0512,00,01,00000000	; [044] 05-12, Terminal 27, 0 - No Operation
0513,00,01,00000000	; [045] 05-13, Terminal 29, 0 - No Operation
0514,00,01,00000004	; [046] 05-14, Terminal 32, 4 - Quick Stop
0510,00,01,00000000	; [047] 05-10, Terminal 18, 0 - No Operation
0175,00,02,00000015	; [048] 01-75, Start Speed, 1,5 Hz
0222,00,02,00000005	; [049] 02-22, Activate Brake Speed ?en bei 0,5 Hz
0124,00,04,00000750	; [050] 01-24, Motor current 7.5 A
0341,00,04,00000100	; [051] 03-41, Ramp 1 ramp up time (1 Sec to 50 Hz)
0342,00,04,00000100	; [052] 03-42, Ramp 1 ramp down time (1 Sec to  0 Hz)
0414,00,02,00001000	; [053] 04-14, Motor Speed High Limit 100,0 Hz
0220,00,04,00000260	; [054] 02-20, Release brake current 2,6 A
(*0130,00,04,00029763	; [---] 01-30, Stator resistance (Rs) 2,9763 Ohm
0131,00,04,00022212	; [---] 01-31, Rotor resistance (Rr) 2,2212 Ohm*)
(*0134,00,04,00031036	; [---] 01-34, Rotor leakage reactance (X2) 3,1036 Ohm*)
;0136,00,04,01803904	; [---] 01-36, Iron loss resistance (Rfe) 1803,904 Ohm
;0135,00,04,00653996	; [---] 01-35, Main reactance (Xh) 65,3996 Ohm
0416,00,02,00002500	; [055] 04-16, Torque limit motor mode, 160,0 - % NOW 250%
0417,00,02,00001600	; [056] 04-17, Torque limit generator mode, 160,0 %
;0133,00,04,00031036	; [---] 01-33, Stator leakage reactance (X1), 3,1036 Ohm
0303,00,04,00100000	; [057] 03-03, Maximum Reference, 100,000
0418,00,04,00002100	; [058] 04-18, Current Limit 172,0 % - NOW 210%
0851,00,01,00000003	; [0] 08-51, Quick stop Logical OR
```

### Data object Logical/Robo_Drive_Control/Param_2_2kwStar (Simple, version 4.00.0) - Parameters 2.2kW Star

#### Param_2_2kwStar.dat
```
(********************************************************************
 * COPYRIGHT --
 ********************************************************************
 * Data object: Param_2kwStar
 * File: Param_2kwStar.dat
 * Author:  D.Jefferys
 * Created: February 12, 2009
 ********************************************************************
 * Data object file: Param_2kwStar.dat
 ********************************************************************)

;Version 2.00 18/10/2010 D.J. Added 14-26 Trip Delay - Disabled, Changed 14-10 from 3 (Coasting) to 5 (Kenetic Backup + Trip)
;Version 3.00 03/11/2010 D.J. Added CAN Switch Settings
;Version 4.00 02/11/2011 D.J. Added Parameter 40 - Hand on Key on LCP now Disabled

;CAN Module Switch Settings
;--------------------------

;Baudrate
;8 on  7 on  Par 10-01
;8 on  7 off 500kbps
;8 off 7 on  250kbps
;8 off 7 off 125kbps

;Node Number Binary
;1 = 1s
;2 = 2s
;3 = 4s
;4 = 8s
;5 = 16s
;6 = 32s

;
;	!!! DO NOT CHANGE THE SEQUENCE OF THE PARAMETERS
;
; FU parameter to the Ubertragung (only parameter, which deviates from the default values)
;
; 2.2 kW Star
;
; Index, Subindex, Datatype (Bytes), Setting (DINT) ; Comments
0002,00,01,00000001	; [000] 00-02, Motor Speed 0 - RPM, 1 - Hz
0001,00,01,00000000	; [001] 00-01, Language 0 - English, 1 - German
0011,00,01,00000001	; [002] 00-11, Edit Setup 1
0190,00,01,00000002	; [003] 01-90, Motor Thermal Protection, 2 - Thermistor
0040,00,01,00000000 ; [---] 00-40, Hand On Key on LCP 0 - Disabled No Function
0381,00,04,00000050 ; [000] 03-81, QuickStop ramp time 100 - 1s
0458,00,01,00000001	; [004] 04-58, Missing motor phase function, 1 - Trip 100ms
0854,00,01,00000001	; [005] 08-54, Reversing select 1 - Bus only 3 - Bus and Terminal
0211,00,02,00000120	; [006] 02-11, Brake resistor 120 Ohm
0212,00,04,00001200	; [007] 02-12, Brake power limit 1200 Watt
0213,00,01,00000002	; [008] 02-13, Brake check 2 - Alarm
1426,00,01,00000000 ; [---] 14-26, Trip delay at inverter fault 0 = Disabled
0803,00,04,00000002 ; [000] 08-03, Control Word Timeout Time 10 = 1Sec
0804,00,01,00000002	; [009] 08-04, Control Word Timeout Function 2 - Stop with auto restart
0801,00,01,00000002	; [010] 08-01, Control Site, 2 - Controlword only
0223,00,01,00000005	; [011] 02-23, Active brake delay 0,3 s
1761,00,01,00000002	; [012] 17-61, Encoder Signal Monitoring (Encoder faulty), 2 - Trip
1710,00,01,00000001	; [013] 17-10, Encoder Signal Type 1 - TTL
1711,00,02,00001024	; [014] 17-11, Encoder Resolution 1024 Pulse
0430,00,01,00000001 ; [015] 04-30, Motor Feedback Loss Function, 1 - Warning, 2* - Trip
0431,00,02,00000300 ; [016] 04-31, Motor Feedback Speed Error RPM, 0-600, 300*
0226,00,02,00005000	; [015] 02-26, Torque Ref, 50,00%
0228,00,02,00000200	; [016] 02-28, Gain Boost Factor, 2,00% 0-4% ***************************
0519,00,01,00000003	; [017] 05-19, Terminal 37 Safe Stop, 3 - Safe Stop Warning
0120,00,04,00000220	; [018] 01-20, Motor Power 2.2kW
0101,00,01,00000003	; [019] 01-01, Motor Control Principle, 3 - Flux with motor feedback
0122,00,02,00000400	; [020] 01-22, Motor voltage 400 V
0123,00,02,00000050	; [021] 01-23, Motor frequency 50 Hz
0162,00,02,00000100	; [022] 01-62, Slip compenstation 100%
0410,00,01,00000002	; [023] 04-10, Motor speed direction, 2 - both directions
0540,00,01,00000032	; [024] 05-40, [0] Relay 1 Function, 32 - Mech brake ctrl
0540,01,01,00000032	; [025] 05-40, [1] Relay 2 Function, 32 - Mech brake ctrl
0802,00,01,00000003 ; [---] 08-02, Control Site 3 - Option A CAN Bus
0102,00,01,00000002	; [026] 01-02, Flux Motor Feeback Source 2 - MCB102
0125,00,02,00001400	; [027] 01-25, Motor nominal speed 1440 rpm
0702,00,02,00000070	; [028] 07-02, Speed PID proportionl gain 0,070
0700,00,01,00000002	; [029] 07-00, Speed PID Feedback Source 2 - MCB102
0172,00,01,00000006	; [030] 01-72, Start function, 6 - Hoist Mech. Brake Rel
0210,00,01,00000001	; [031] 02-10, Brake Function, 1 - Resistor brake
1410,00,01,00000005	; [032] 14-10, Mains failure, 3 - Coasting 5 - Kenetic backup , trip
0193,00,01,00000006	; [033] 01-93, Thermistor source, 6 - Digital Input 33
0100,00,01,00000001	; [034] 01-00, Configuration mode, 1 - Closed loop with encoder
0139,00,01,00000004	; [035] 01-39, Motor poles, 4
0511,00,01,00000000	; [036] 05-11, Terminal 19, 0 - No Operation
0512,00,01,00000000	; [037] 05-12, Terminal 27, 0 - No Operation
0513,00,01,00000000	; [038] 05-13, Terminal 29, 0 - No Operation
0510,00,01,00000000	; [039] 05-10, Terminal 18, 0 - No Operation
0175,00,02,00000015	; [040] 01-75, Start Speed, 1,5 Hz
0222,00,02,00000005	; [041] 02-22, Activate Brake Speed ?en bei 0,5 Hz
0124,00,04,00000520	; [042] 01-24, Motor current 5,2 A
0341,00,04,00000100	; [043] 03-41, Ramp 1 ramp up time (1 Sec to 50 Hz)
0342,00,04,00000100	; [044] 03-42, Ramp 1 ramp down time (1 Sec to  0 Hz)
0414,00,02,00001000	; [045] 04-14, Motor Speed High Limit 100,0 Hz
0220,00,04,00000260	; [046] 02-20, Release brake current 2,6 A
0130,00,04,00029763	; [047] 01-30, Stator resistance (Rs) 2,9763 Ohm
0131,00,04,00022212	; [048] 01-31, Rotor resistance (Rr) 2,2212 Ohm
0134,00,04,00031036	; [049] 01-34, Rotor leakage reactance (X2) 3,1036 Ohm
;0136,00,04,01803904	; [050] 01-36, Iron loss resistance (Rfe) 1803,904 Ohm
;0135,00,04,00653996	; [051] 01-35, Main reactance (Xh) 65,3996 Ohm
0416,00,02,00002500	; [052] 04-16, Torque limit motor mode, 160,0 - % NOW 250%
0417,00,02,00001600	; [053] 04-17, Torque limit generator mode, 160,0 %
;0133,00,04,00031036	; [054] 01-33, Stator leakage reactance (X1), 3,1036 Ohm
0303,00,04,00100000	; [055] 03-03, Maximum Reference, 100,000
0418,00,04,00002500	; [056] 04-18, Current Limit 172,0 % - NOW 250%
```

### Data object Logical/Robo_Drive_Control/ParamD15 (Simple, version 4.00.0) - Parameters 1.5kW Star Disable Drive feedback

#### ParamD15.dat
```
(********************************************************************
 * COPYRIGHT --
 ********************************************************************
 * Data object: Param_1_5kwStar
 * File: Param_1_5kwStar.dat
 * Author:  D.Jefferys
 * Created: October 2, 2009
 ********************************************************************
 * Data object file: Param_1_5kwStar.dat
 ********************************************************************)

;Version 2.00 18/10/2010 D.J. Added 14-26 Trip Delay - Disabled, Changed 14-10 from 3 (Coasting) to 5 (Kenetic Backup + Trip)
;Version 3.00 03/11/2010 D.J. Added CAN Switch Settings
;Version 4.00 02/11/2011 D.J. Added Parameter 40 - Hand on Key on LCP now Disabled

;CAN Module Switch Settings
;--------------------------

;Baudrate
;8 on  7 on  Par 10-01
;8 on  7 off 500kbps
;8 off 7 on  250kbps
;8 off 7 off 125kbps

;Node Number Binary
;1 = 1s
;2 = 2s
;3 = 4s
;4 = 8s
;5 = 16s
;6 = 32s

;
;	!!! DO NOT CHANGE THE SEQUENCE OF THE PARAMETERS
;
; FU parameter to the Ubertragung (only parameter, which deviates from the default values)
;
; 1.5 kW Star
;
; Index, Subindex, Datatype (Bytes), Setting (DINT) ; Comments
0002,00,01,00000001	; [000] 00-02, Motor Speed 0 - RPM, 1 - Hz
0001,00,01,00000000	; [001] 00-01, Language 0 - English, 1 - German
0011,00,01,00000001	; [002] 00-11, Edit Setup 1
0190,00,01,00000000	; [003] 01-90, Motor Thermal Protection, 2 - Thermistor
0040,00,01,00000000 ; [---] 00-40, Hand On Key on LCP 0 - Disabled No Function
0381,00,04,00000050 ; [000] 03-81, QuickStop ramp time 100 - 1s
0458,00,01,00000001	; [004] 04-58, Missing motor phase function, 1 - Trip 100ms
0854,00,01,00000001	; [005] 08-54, Reversing select 1 - Bus only 3 - Bus and Terminal
0211,00,02,00000310	; [006] 02-11, Brake resistor 120 Ohm
0212,00,04,00001200	; [007] 02-12, Brake power limit 1200 Watt
0213,00,01,00000002	; [008] 02-13, Brake check 2 - Alarm
1426,00,01,00000000 ; [---] 14-26, Trip delay at inverter fault 0 = Disabled
0803,00,04,00000002 ; [000] 08-03, Control Word Timeout Time 10 = 1Sec
0804,00,01,00000002	; [009] 08-04, Control Word Timeout Function 2 - Stop with auto restart
0801,00,01,00000002	; [010] 08-01, Control Site, 2 - Controlword only
0223,00,01,00000005	; [011] 02-23, Active brake delay 0,3 s
1761,00,01,00000000	;********************** [012] 17-61, Encoder Signal Monitoring (Encoder faulty), 2 - Trip Changed for testing.
1710,00,01,00000001	; [013] 17-10, Encoder Signal Type 1 - TTL
1711,00,02,00001024	; [014] 17-11, Encoder Resolution 1024 Pulse
0430,00,01,00000001 ; [015] 04-30, Motor Feedback Loss Function, 1 - Warning, 2* - Trip
0431,00,02,00000300 ; [016] 04-31, Motor Feedback Speed Error RPM, 0-600, 300*
0226,00,02,00005000	; [015] 02-26, Torque Ref, 50,00%
0228,00,02,00000200	; [016] 02-28, Gain Boost Factor, 2,00% 0-4% ***************************
0519,00,01,00000003	; [017] 05-19, Terminal 37 Safe Stop, 3 - Safe Stop Warning
0120,00,04,00000150	; [018] 01-20, Motor Power 1.5kW
0101,00,01,00000003	; [019] 01-01, Motor Control Principle, 3 - Flux with motor feedback
0122,00,02,00000400	; [020] 01-22, Motor voltage 400 V
0123,00,02,00000050	; [021] 01-23, Motor frequency 50 Hz
0162,00,02,00000100	; [022] 01-62, Slip compenstation 100%
0410,00,01,00000002	; [023] 04-10, Motor speed direction, 2 - both directions
0540,00,01,00000032	; [024] 05-40, [0] Relay 1 Function, 32 - Mech brake ctrl
0540,01,01,00000032	; [025] 05-40, [1] Relay 2 Function, 32 - Mech brake ctrl
0802,00,01,00000003 ; [---] 08-02, Control Site 3 - Option A CAN Bus
0102,00,01,00000002	; [026] 01-02, Flux Motor Feeback Source 2 - MCB102
0125,00,02,00001400	; [027] 01-25, Motor nominal speed 1440 rpm
0702,00,02,00000070	; [028] 07-02, Speed PID proportionl gain 0,070
0700,00,01,00000002	; [029] 07-00, Speed PID Feedback Source 2 - MCB102
0172,00,01,00000006	; [030] 01-72, Start function, 6 - Hoist Mech. Brake Rel
0210,00,01,00000001	; [031] 02-10, Brake Function, 1 - Resistor brake
1410,00,01,00000005	; [032] 14-10, Mains failure, 3 - Coasting 5 - Kenetic backup , trip
0193,00,01,00000006	; [033] 01-93, Thermistor source, 6 - Digital Input 33
0100,00,01,00000001	; [034] 01-00, Configuration mode, 1 - Closed loop with encoder
0139,00,01,00000004	; [035] 01-39, Motor poles, 4
0511,00,01,00000000	; [036] 05-11, Terminal 19, 0 - No Operation
0512,00,01,00000000	; [037] 05-12, Terminal 27, 0 - No Operation
0513,00,01,00000000	; [038] 05-13, Terminal 29, 0 - No Operation
0510,00,01,00000000	; [039] 05-10, Terminal 18, 0 - No Operation
0175,00,02,00000015	; [040] 01-75, Start Speed, 1,5 Hz
0222,00,02,00000005	; [041] 02-22, Activate Brake Speed ?en bei 0,5 Hz
0124,00,04,00000360	; [042] 01-24, Motor current 5,2 A
0341,00,04,00000100	; [043] 03-41, Ramp 1 ramp up time (1 Sec to 50 Hz)
0342,00,04,00000100	; [044] 03-42, Ramp 1 ramp down time (1 Sec to  0 Hz)
0414,00,02,00001000	; [045] 04-14, Motor Speed High Limit 100,0 Hz
0220,00,04,00000180	; [046] 02-20, Release brake current 1,8 A - About Half of motor A?
;0130,00,04,00029763	; [047] 01-30, Stator resistance (Rs) 2,9763 Ohm
;0131,00,04,00022212	; [048] 01-31, Rotor resistance (Rr) 2,2212 Ohm
;0134,00,04,00031036	; [049] 01-34, Rotor leakage reactance (X2) 3,1036 Ohm
;0136,00,04,01803904	; [050] 01-36, Iron loss resistance (Rfe) 1803,904 Ohm
;0135,00,04,00653996	; [051] 01-35, Main reactance (Xh) 65,3996 Ohm
0416,00,02,00002500	; [052] 04-16, Torque limit motor mode, 160,0 - % NOW 250%
0417,00,02,00001600	; [053] 04-17, Torque limit generator mode, 160,0 %
;0133,00,04,00031036	; [054] 01-33, Stator leakage reactance (X1), 3,1036 Ohm
0303,00,04,00100000	; [055] 03-03, Maximum Reference, 100,000
0418,00,04,00001720	; [056] 04-18, Current Limit 172,0 % - NOW 250%
```

### Data object Logical/Robo_Drive_Control/Param_1_5kwStar_expo (Simple, version 4.00.0) - Parameters 1.5kW Star

#### Param_1_5kwStar.dat
```
(********************************************************************
 * COPYRIGHT --
 ********************************************************************
 * Data object: Param_1_5kwStar
 * File: Param_1_5kwStar.dat
 * Author:  D.Jefferys
 * Created: October 2, 2009
 ********************************************************************
 * Data object file: Param_1_5kwStar.dat
 ********************************************************************)

;Version 2.00 18/10/2010 D.J. Added 14-26 Trip Delay - Disabled, Changed 14-10 from 3 (Coasting) to 5 (Kenetic Backup + Trip)
;Version 3.00 03/11/2010 D.J. Added CAN Switch Settings
;Version 4.00 02/11/2011 D.J. Added Parameter 40 - Hand on Key on LCP now Disabled

;CAN Module Switch Settings
;--------------------------

;Baudrate
;8 on  7 on  Par 10-01
;8 on  7 off 500kbps
;8 off 7 on  250kbps
;8 off 7 off 125kbps

;Node Number Binary
;1 = 1s
;2 = 2s
;3 = 4s
;4 = 8s
;5 = 16s
;6 = 32s

;
;	!!! DO NOT CHANGE THE SEQUENCE OF THE PARAMETERS
;
; FU parameter to the Ubertragung (only parameter, which deviates from the default values)
;
; 1.5 kW Star
;
; Index, Subindex, Datatype (Bytes), Setting (DINT) ; Comments
0002,00,01,00000001	; [000] 00-02, Motor Speed 0 - RPM, 1 - Hz
0001,00,01,00000000	; [001] 00-01, Language 0 - English, 1 - German
0011,00,01,00000001	; [002] 00-11, Edit Setup 1
0190,00,01,00000000	; [003] 01-90, Motor Thermal Protection, 2 - Thermistor
0040,00,01,00000000 ; [---] 00-40, Hand On Key on LCP 0 - Disabled No Function
0381,00,04,00000050 ; [000] 03-81, QuickStop ramp time 100 - 1s
0458,00,01,00000001	; [004] 04-58, Missing motor phase function, 1 - Trip 100ms
0854,00,01,00000001	; [005] 08-54, Reversing select 1 - Bus only 3 - Bus and Terminal
0211,00,02,00000310	; [006] 02-11, Brake resistor 120 Ohm
0212,00,04,00001200	; [007] 02-12, Brake power limit 1200 Watt
0213,00,01,00000002	; [008] 02-13, Brake check 2 - Alarm
1426,00,01,00000000 ; [---] 14-26, Trip delay at inverter fault 0 = Disabled
0803,00,04,00000002 ; [000] 08-03, Control Word Timeout Time 10 = 1Sec
0804,00,01,00000002	; [009] 08-04, Control Word Timeout Function 2 - Stop with auto restart
0801,00,01,00000002	; [010] 08-01, Control Site, 2 - Controlword only
0223,00,01,00000005	; [011] 02-23, Active brake delay 0,3 s
1761,00,01,00000002	; [012] 17-61, Encoder Signal Monitoring (Encoder faulty), 2 - Trip Changed for testing.
1710,00,01,00000001	; [013] 17-10, Encoder Signal Type 1 - TTL
1711,00,02,00001024	; [014] 17-11, Encoder Resolution 1024 Pulse
0430,00,01,00000001 ; [015] 04-30, Motor Feedback Loss Function, 1 - Warning, 2* - Trip
0431,00,02,00000300 ; [016] 04-31, Motor Feedback Speed Error RPM, 0-600, 300*
0226,00,02,00005000	; [015] 02-26, Torque Ref, 50,00%
0228,00,02,00000200	; [016] 02-28, Gain Boost Factor, 2,00% 0-4% ***************************
0519,00,01,00000003	; [017] 05-19, Terminal 37 Safe Stop, 3 - Safe Stop Warning
0120,00,04,00000150	; [018] 01-20, Motor Power 1.5kW
0101,00,01,00000003	; [019] 01-01, Motor Control Principle, 3 - Flux with motor feedback
0122,00,02,00000400	; [020] 01-22, Motor voltage 400 V
0123,00,02,00000050	; [021] 01-23, Motor frequency 50 Hz
0162,00,02,00000100	; [022] 01-62, Slip compenstation 100%
0410,00,01,00000002	; [023] 04-10, Motor speed direction, 2 - both directions
0540,00,01,00000032	; [024] 05-40, [0] Relay 1 Function, 32 - Mech brake ctrl
0540,01,01,00000032	; [025] 05-40, [1] Relay 2 Function, 32 - Mech brake ctrl
0802,00,01,00000003 ; [---] 08-02, Control Site 3 - Option A CAN Bus
0102,00,01,00000002	; [026] 01-02, Flux Motor Feeback Source 2 - MCB102
0125,00,02,00001400	; [027] 01-25, Motor nominal speed 1440 rpm
0702,00,02,00000070	; [028] 07-02, Speed PID proportionl gain 0,070
0700,00,01,00000002	; [029] 07-00, Speed PID Feedback Source 2 - MCB102
0172,00,01,00000006	; [030] 01-72, Start function, 6 - Hoist Mech. Brake Rel
0210,00,01,00000001	; [031] 02-10, Brake Function, 1 - Resistor brake
1410,00,01,00000005	; [032] 14-10, Mains failure, 3 - Coasting 5 - Kenetic backup , trip
0193,00,01,00000006	; [033] 01-93, Thermistor source, 6 - Digital Input 33
0100,00,01,00000001	; [034] 01-00, Configuration mode, 1 - Closed loop with encoder
0139,00,01,00000004	; [035] 01-39, Motor poles, 4
0511,00,01,00000000	; [036] 05-11, Terminal 19, 0 - No Operation
0512,00,01,00000000	; [037] 05-12, Terminal 27, 0 - No Operation
0513,00,01,00000000	; [038] 05-13, Terminal 29, 0 - No Operation
0510,00,01,00000000	; [039] 05-10, Terminal 18, 0 - No Operation
0175,00,02,00000015	; [040] 01-75, Start Speed, 1,5 Hz
0222,00,02,00000005	; [041] 02-22, Activate Brake Speed ?en bei 0,5 Hz
0124,00,04,00000360	; [042] 01-24, Motor current 5,2 A
0341,00,04,00000100	; [043] 03-41, Ramp 1 ramp up time (1 Sec to 50 Hz)
0342,00,04,00000100	; [044] 03-42, Ramp 1 ramp down time (1 Sec to  0 Hz)
0414,00,02,00001000	; [045] 04-14, Motor Speed High Limit 100,0 Hz
0220,00,04,00000180	; [046] 02-20, Release brake current 1,8 A - About Half of motor A?
;0130,00,04,00029763	; [047] 01-30, Stator resistance (Rs) 2,9763 Ohm
;0131,00,04,00022212	; [048] 01-31, Rotor resistance (Rr) 2,2212 Ohm
;0134,00,04,00031036	; [049] 01-34, Rotor leakage reactance (X2) 3,1036 Ohm
;0136,00,04,01803904	; [050] 01-36, Iron loss resistance (Rfe) 1803,904 Ohm
;0135,00,04,00653996	; [051] 01-35, Main reactance (Xh) 65,3996 Ohm
0416,00,02,00002500	; [052] 04-16, Torque limit motor mode, 160,0 - % NOW 250%
0417,00,02,00001600	; [053] 04-17, Torque limit generator mode, 160,0 %
;0133,00,04,00031036	; [054] 01-33, Stator leakage reactance (X1), 3,1036 Ohm
0303,00,04,00100000	; [055] 03-03, Maximum Reference, 100,000
0418,00,04,00001720	; [056] 04-18, Current Limit 172,0 % - NOW 250%
```

### Data object Logical/Robo_Drive_Control/Param_0_25kwStar1 (Simple, version 4.00.0) - Parameters 0.25kW Star

#### Param_0_25kwStar.dat
```
(********************************************************************
 * COPYRIGHT --
 ********************************************************************
 * Data object: Param_2kwStar
 * File: Param_2kwStar.dat
 * Author:  D.Jefferys
 * Created: February 12, 2009
 ********************************************************************
 * Data object file: Param_2kwStar.dat
 ********************************************************************)

;Version 2.00 18/10/2010 D.J. Added 14-26 Trip Delay - Disabled, Changed 14-10 from 3 (Coasting) to 5 (Kenetic Backup + Trip)
;Version 3.00 03/11/2010 D.J. Added CAN Switch Settings
;Version 4.00 02/11/2011 D.J. Added Parameter 40 - Hand on Key on LCP now Disabled

;CAN Module Switch Settings
;--------------------------

;Baudrate
;8 on  7 on  Par 10-01
;8 on  7 off 500kbps
;8 off 7 on  250kbps
;8 off 7 off 125kbps

;Node Number Binary
;1 = 1s
;2 = 2s
;3 = 4s
;4 = 8s
;5 = 16s
;6 = 32s

;
;	!!! DO NOT CHANGE THE SEQUENCE OF THE PARAMETERS
;
; FU parameter to the Ubertragung (only parameter, which deviates from the default values)
;
; 0.25 kW Star
;
; Index, Subindex, Datatype (Bytes), Setting (DINT) ; Comments
0002,00,01,00000001	; [000] 00-02, Motor Speed 0 - RPM, 1 - Hz
0001,00,01,00000000	; [001] 00-01, Language 0 - English, 1 - German
0011,00,01,00000001	; [002] 00-11, Edit Setup 1
;0190,00,01,00000000	; [003] 01-90, Motor Thermal Protection, 0 - No protection
0040,00,01,00000000 ; [---] 00-40, Hand On Key on LCP 0 - Disabled No Function
0381,00,04,00000050 ; [000] 03-81, QuickStop ramp time 100 - 1s
;0458,00,01,00000001	; [004] 04-58, Missing motor phase function, 1 - Trip 100ms
0854,00,01,00000001	; [005] 08-54, Reversing select 1 - Bus only 3 - Bus and Terminal
0211,00,02,00000620	; [006] 02-11, Brake resistor 620 Ohm
0212,00,04,00000065	; [007] 02-12, Brake power limit 65 Watt
0213,00,01,00000002	; [008] 02-13, Brake check 2 - Alarm
1426,00,01,00000000 ; [---] 14-26, Trip delay at inverter fault 0 = Disabled
0803,00,04,00000002 ; [000] 08-03, Control Word Timeout Time 10 = 1Sec
0804,00,01,00000002	; [009] 08-04, Control Word Timeout Function 2 - Stop with auto restart
0801,00,01,00000002	; [010] 08-01, Control Site, 2 - Controlword only
0223,00,01,00000005	; [011] 02-23, Active brake delay 0,3 s
1761,00,01,00000002	; [012] 17-61, Encoder Signal Monitoring (Encoder faulty), 2 - Trip
1710,00,01,00000001	; [013] 17-10, Encoder Signal Type 1 - TTL
1711,00,02,00001024	; [014] 17-11, Encoder Resolution 1024 Pulse
0430,00,01,00000001 ; [015] 04-30, Motor Feedback Loss Function, 1 - Warning, 2* - Trip
0431,00,02,00000600 ; [016] 04-31, Motor Feedback Speed Error RPM, 0-600, 300*
0226,00,02,00005000	; [017] 02-26, Torque Ref, 50,00%
0228,00,02,00000200	; [018] 02-28, Gain Boost Factor, 2,00% 0-4% ***************************
0519,00,01,00000003	; [019] 05-19, Terminal 37 Safe Stop, 3 - Safe Stop Warning
0120,00,04,00000025	; [020] 01-20, Motor Power 0.25kW
0101,00,01,00000003	; [021] 01-01, Motor Control Principle, 3 - Flux with motor feedback
0122,00,02,00000400	; [022] 01-22, Motor voltage 400 V
0123,00,02,00000050	; [023] 01-23, Motor frequency 50 Hz
0162,00,02,00000100	; [024] 01-62, Slip compenstation 100%
0410,00,01,00000002	; [025] 04-10, Motor speed direction, 2 - both directions
0540,00,01,00000032	; [026] 05-40, [0] Relay 1 Function, 32 - Mech brake ctrl
0540,01,01,00000032	; [027] 05-40, [1] Relay 2 Function, 32 - Mech brake ctrl
0802,00,01,00000003 ; [---] 08-02, Control Site 3 - Option A CAN Bus
0102,00,01,00000002	; [028] 01-02, Flux Motor Feeback Source 2 - MCB102
0125,00,02,00001350	; [029] 01-25, Motor nominal speed 1350 rpm
0702,00,02,00000040	; [030] 07-02, Speed PID proportionl gain 0,040
0700,00,01,00000002	; [031] 07-00, Speed PID Feedback Source 2 - MCB102
0172,00,01,00000006	; [032] 01-72, Start function, 6 - Hoist Mech. Brake Rel
0210,00,01,00000001	; [033] 02-10, Brake Function, 1 - Resistor brake
1410,00,01,00000005	; [034] 14-10, Mains failure, 3 - Coasting 5 - Kenetic backup , trip
;0193,00,01,00000006	; [035] 01-93, Thermistor source, 6 - Digital Input 33
0100,00,01,00000001	; [036] 01-00, Configuration mode, 1 - Closed loop with encoder
0139,00,01,00000004	; [037] 01-39, Motor poles, 4
0511,00,01,00000000	; [038] 05-11, Terminal 19, 0 - No Operation
0512,00,01,00000000	; [039] 05-12, Terminal 27, 0 - No Operation
0513,00,01,00000000	; [040] 05-13, Terminal 29, 0 - No Operation
0510,00,01,00000000	; [041] 05-10, Terminal 18, 0 - No Operation
0175,00,02,00000015	; [042] 01-75, Start Speed, 1,5 Hz
0222,00,02,00000005	; [043] 02-22, Activate Brake Speed ?en bei 0,5 Hz
0124,00,04,00000089	; [044] 01-24, Motor current 0,89 A
0341,00,04,00000100	; [045] 03-41, Ramp 1 ramp up time (1 Sec to 50 Hz)
0342,00,04,00000100	; [046] 03-42, Ramp 1 ramp down time (1 Sec to  0 Hz)
0414,00,02,00001000	; [047] 04-14, Motor Speed High Limit 100,0 Hz
;0220,00,04,00000260	; [048] 02-20, Release brake current 2,6 A
;0130,00,04,00029763	; [049] 01-30, Stator resistance (Rs) 2,9763 Ohm
;0131,00,04,00022212	; [050] 01-31, Rotor resistance (Rr) 2,2212 Ohm
;0132,00,04,00031036	; [051] 01-34, Rotor leakage reactance (X2) 3,1036 Ohm
;0136,00,04,01803904	; [052] 01-36, Iron loss resistance (Rfe) 1803,904 Ohm
;0135,00,04,00653996	; [053] 01-35, Main reactance (Xh) 65,3996 Ohm
0416,00,02,00001600	; [054] 04-16, Torque limit motor mode, 160,0 %
0417,00,02,00001600	; [055] 04-17, Torque limit generator mode, 160,0 %
;0133,00,04,00031036	; [056] 01-33, Stator leakage reactance (X1), 3,1036 Ohm
0303,00,04,00050000	; [057] 03-03, Maximum Reference, 100,000 50,000 Rotate for now!
0418,00,04,00001720	; [058] 04-18, Current Limit 172,0 %
```

### Data object Logical/Robo_Drive_Control/ParaTest (Simple) - Parameters 0.25kW Test No Feed Back

#### ParaTest.dat
```
(********************************************************************
 * COPYRIGHT --
 ********************************************************************
 * Data object: ParaTest
 * File: ParaTest.dat
 * Author:  D.Jefferys
 * Created: February 12, 2009
 ********************************************************************
 * Data object file: ParaTest.dat
 ********************************************************************)

 ;
;	!!! DO NOT CHANGE THE SEQUENCE OF THE PARAMETERS
;
; FU parameter to the Ubertragung (only parameter, which deviates from the default values)
;
; 0.25 kW Star
;
; Index, Subindex, Datatype (Bytes), Setting (DINT) ; Comments
;;;0002,00,01,00000001	; [000] 00-02, Motor Speed 0 - RPM, 1 - Hz
0001,00,01,00000000	; [001] 00-01, Language 0 - English, 1 - German
0011,00,01,00000001	; [002] 00-11, Edit Setup 1
;0190,00,01,00000002	; [003] 01-90, Motor Thermal Protection, 2 - Thermistor
0381,00,04,00000045 ; [000] 03-81, QuickStop ramp time 100 - 1s
0458,00,01,00000001	; [004] 04-58, Missing motor phase function, 1 - Trip 100ms
0854,00,01,00000001	; [005] 08-54, Reversing select 1 - Bus only 3 - Bus and Terminal
;0211,00,02,00000620	; [006] 02-11, Brake resistor 620 Ohm
;0212,00,04,00000065	; [007] 02-12, Brake power limit 65 Watt
;0213,00,01,00000002	; [008] 02-13, Brake check 2 - Alarm
0803,00,04,00000002 ; [000] 08-03, Control Word Timeout Time 10 = 1Sec
0804,00,01,00000002	; [009] 08-04, Control Word Timeout Function 2 - Stop with auto restart
0801,00,01,00000002	; [010] 08-01, Control Site, 2 - Controlword only
0223,00,01,00000005	; [011] 02-23, Active brake delay 0,3 s
;1761,00,01,00000002	; [012] 17-61, Encoder Signal Monitoring (Encoder faulty), 2 - Trip
;1710,00,01,00000001	; [013] 17-10, Encoder Signal Type 1 - TTL
;1711,00,02,00001024	; [014] 17-11, Encoder Resolution 1024 Pulse
;0430,00,01,00000001 ; [015] 04-30, Motor Feedback Loss Function, 1 - Warning, 2* - Trip
;0431,00,02,00000600 ; [016] 04-31, Motor Feedback Speed Error RPM, 0-600, 300*
;;;0226,00,02,00005000	; [015] 02-26, Torque Ref, 50,00%
;;;0228,00,02,00000200	; [016] 02-28, Gain Boost Factor, 2,00% 0-4% ***************************
;;;0519,00,01,00000003	; [017] 05-19, Terminal 37 Safe Stop, 3 - Safe Stop Warning
0120,00,04,00000025	; [018] 01-20, Motor Power 0.25kW
;0101,00,01,00000003	; [019] 01-01, Motor Control Principle, 3 - Flux with motor feedback
0122,00,02,00000230	; [020] 01-22, Motor voltage 400 V
0123,00,02,00000050	; [021] 01-23, Motor frequency 50 Hz
;;;0162,00,02,00000100	; [022] 01-62, Slip compenstation 100%
0410,00,01,00000002	; [023] 04-10, Motor speed direction, 2 - both directions
0540,00,01,00000032	; [024] 05-40, [0] Relay 1 Function, 32 - Mech brake ctrl
0540,01,01,00000032	; [025] 05-40, [1] Relay 2 Function, 32 - Mech brake ctrl
0802,00,01,00000003 ; [---] 08-02, Control Site 3 - Option A CAN Bus
;0102,00,01,00000002	; [026] 01-02, Flux Motor Feeback Source 2 - MCB102
;0125,00,02,00001400	; [027] 01-25, Motor nominal speed 1440 rpm
;0702,00,02,00000070	; [028] 07-02, Speed PID proportionl gain 0,070
;0700,00,01,00000002	; [029] 07-00, Speed PID Feedback Source 2 - MCB102
;;;0172,00,01,00000006	; [030] 01-72, Start function, 6 - Hoist Mech. Brake Rel
;0210,00,01,00000001	; [031] 02-10, Brake Function, 1 - Resistor brake
;;;1410,00,01,00000003	; [032] 14-10, Mains failure, 3 - Motorfreilauf
;0193,00,01,00000006	; [033] 01-93, Thermistor source, 6 - Digital Input 33
;0100,00,01,00000001	; [034] 01-00, Configuration mode, 1 - Closed loop with encoder
;0139,00,01,00000004	; [035] 01-39, Motor poles, 4
0511,00,01,00000000	; [036] 05-11, Terminal 19, 0 - No Operation
0512,00,01,00000000	; [037] 05-12, Terminal 27, 0 - No Operation
0513,00,01,00000000	; [038] 05-13, Terminal 29, 0 - No Operation
0510,00,01,00000000	; [039] 05-10, Terminal 18, 0 - No Operation
;0175,00,02,00000000	; [040] 01-75, Start Speed, 1,5 Hz
;0222,00,02,00000000	; [041] 02-22, Activate Brake Speed ?en bei 0,5 Hz
0124,00,04,00000139	; [042] 01-24, Motor current 1.39 A
0341,00,04,00000100	; [043] 03-41, Ramp 1 ramp up time (1 Sec to 50 Hz)
0342,00,04,00000100	; [044] 03-42, Ramp 1 ramp down time (1 Sec to  0 Hz)
;;;0414,00,02,00001000	; [045] 04-14, Motor Speed High Limit 100,0 Hz
;0220,00,04,00000260	; [046] 02-20, Release brake current 2,6 A
;0130,00,04,000105080	; [047] 01-30, Stator resistance (Rs) 10.5086 Ohm
;0131,00,04,00022212	; [048] 01-31, Rotor resistance (Rr) 2,2212 Ohm
;0132,00,04,00031036	; [049] 01-34, Rotor leakage reactance (X2) 3,1036 Ohm
;0136,00,04,01803904	; [050] 01-36, Iron loss resistance (Rfe) 1803,904 Ohm
;0135,00,04,00653996	; [051] 01-35, Main reactance (Xh) 65,3996 Ohm
;0416,00,02,00001600	; [052] 04-16, Torque limit motor mode, 160,0 %
;0417,00,02,00001600	; [053] 04-17, Torque limit generator mode, 160,0 %
;0133,00,04,00031036	; [054] 01-33, Stator leakage reactance (X1), 3,1036 Ohm
;0303,00,04,00100000	; [055] 03-03, Maximum Reference, 100,000
0418,00,04,00001720	; [056] 04-18, Current Limit 172,0 %
```

### Program Logical/Robo_Drive_Control/zzRoboPosnNames (IEC) - Robo Position Names - Transfer TrackView

#### zzRoboPosnNames.ab - Implementation code
```automation-basic
(********************************************************************
 * COPYRIGHT -- HP
 ********************************************************************
 * Program: zzRoboPosnNames
 * File: zzRoboPosnNames.ab
 * Author: Dave
 * Created: January 28, 2013
 ********************************************************************
 * Implementation of program zzRoboPosnNames
 ********************************************************************)

PROGRAM _INIT

(* TODO : Add your code here *)

END_PROGRAM

PROGRAM _CYCLIC

	myTviewRobo = D[90]
	myTviewPosn = D[91]

	;New Robo selected then reset current position
	IF (myTviewRobo <> myPLCRobo) THEN
		myPLCRobo = myTviewRobo
		myPLCPosn = 1
	ENDIF

	;Select next position once TrackView has ready the previous
	IF ((myPLCRobo > 0) AND (myTviewPosn = myPLCPosn)) THEN
		IF myPLCPosn < MaxPositions THEN
			myPLCPosn = myPLCPosn + 1
		ENDIF
	ENDIF

	D[92] = myPLCRobo
	D[93] = myPLCPosn
	D[94] = RB_PosnName[myPLCRobo].Name[myPLCPosn]
	D[95] = RB_PosnName[myPLCRobo].Extra[myPLCPosn]

END_PROGRAM
```

#### zzRoboPosnNames.var - Local variables
```iecst
(********************************************************************
 * COPYRIGHT -- HP
 ********************************************************************
 * Program: zzRoboPosnNames
 * File: zzRoboPosnNames.var
 * Author: Dave
 * Created: January 28, 2013
 ********************************************************************
 * Local variables of program zzRoboPosnNames
 ********************************************************************)
VAR
	myTviewRobo : UINT;
	myTviewPosn : UINT;
	myPLCRobo : UINT;
	myPLCPosn : UINT;
END_VAR
```

### Program Logical/Robo_Drive_Control/zzRoboPosnNamesTest (IEC) - Robo Position Names Test

#### zzRoboPosnNamesTest.ab - Implementation code
```automation-basic
(********************************************************************
 * COPYRIGHT -- HP
 ********************************************************************
 * Program: zzRoboPosnNamesTest
 * File: zzRoboPosnNamesTest.ab
 * Author: Dave
 * Created: January 28, 2013
 ********************************************************************
 * Implementation of program zzRoboPosnNamesTest
 ********************************************************************)

PROGRAM _INIT

(* TODO : Add your code here *)

END_PROGRAM

PROGRAM _CYCLIC

;Position Names
myVC = 1
RB_PosnName[myVC].Name[1]	= posnNameHighLevelBagIn
RB_PosnName[myVC].Extra[1]	= posnExtraNone
RB_PosnName[myVC].Name[2]	= posnNameHighLevelBagOut
RB_PosnName[myVC].Extra[2]	= posnExtraNone
RB_PosnName[myVC].Name[3]	= posnNameLowLevelBagOut
RB_PosnName[myVC].Extra[3]	= posnExtraNone
RB_PosnName[myVC].Name[4]	= posnNameLowLevelBagIn
RB_PosnName[myVC].Extra[4]	= posnExtraNone
RB_PosnName[myVC].Name[5]	= posnNameNone
RB_PosnName[myVC].Extra[5]	= posnExtraNone
RB_PosnName[myVC].Name[6]	= posnNameNone
RB_PosnName[myVC].Extra[6]	= posnExtraNone

myVC = 2
RB_PosnName[myVC].Name[1]	= posnNameHighLevelBagIn
RB_PosnName[myVC].Extra[1]	= posnExtraNone
RB_PosnName[myVC].Name[2]	= posnNameHighLevelBagOut
RB_PosnName[myVC].Extra[2]	= posnExtraNone
RB_PosnName[myVC].Name[3]	= posnNameLowLevelBagOut
RB_PosnName[myVC].Extra[3]	= posnExtraNone
RB_PosnName[myVC].Name[4]	= posnNameLowLevelBagIn
RB_PosnName[myVC].Extra[4]	= posnExtraNone
RB_PosnName[myVC].Name[5]	= posnNameNone
RB_PosnName[myVC].Extra[5]	= posnExtraNone
RB_PosnName[myVC].Name[6]	= posnNameNone
RB_PosnName[myVC].Extra[6]	= posnExtraNone

myVC = 3
RB_PosnName[myVC].Name[1]	= posnNameHighLevelBagOut
RB_PosnName[myVC].Extra[1]	= posnExtraNone
RB_PosnName[myVC].Name[2]	= posnNameHighLevelBagIn
RB_PosnName[myVC].Extra[2]	= posnExtraNone
RB_PosnName[myVC].Name[3]	= posnNameLoading
RB_PosnName[myVC].Extra[3]	= posnExtraNone
RB_PosnName[myVC].Name[4]	= posnNameNone
RB_PosnName[myVC].Extra[4]	= posnExtraNone
RB_PosnName[myVC].Name[5]	= posnNameNone
RB_PosnName[myVC].Extra[5]	= posnExtraNone
RB_PosnName[myVC].Name[6]	= posnNameNone
RB_PosnName[myVC].Extra[6]	= posnExtraNone

END_PROGRAM
```

#### zzRoboPosnNamesTest.var - Local variables
```iecst
(********************************************************************
 * COPYRIGHT -- HP
 ********************************************************************
 * Program: zzRoboPosnNamesTest
 * File: zzRoboPosnNamesTest.var
 * Author: Dave
 * Created: January 28, 2013
 ********************************************************************
 * Local variables of program zzRoboPosnNamesTest
 ********************************************************************)
VAR
	myVC : UINT;
END_VAR
```

### Data object Logical/Robo_Drive_Control/Param_1_5kwStar (Simple, version 4.00.1) - Parameters 1.5kW Star

#### Param_1_5kwStar.dat
```
(********************************************************************
 * COPYRIGHT --
 ********************************************************************
 * Data object: Param_1_5kwStar
 * File: Param_1_5kwStar.dat
 * Author:  D.Jefferys
 * Created: October 2, 2009
 ********************************************************************
 * Data object file: Param_1_5kwStar.dat
 ********************************************************************)

;Version 2.00 18/10/2010 D.J. Added 14-26 Trip Delay - Disabled, Changed 14-10 from 3 (Coasting) to 5 (Kenetic Backup + Trip)
;Version 3.00 03/11/2010 D.J. Added CAN Switch Settings
;Version 4.00 02/11/2011 D.J. Added Parameter 40 - Hand on Key on LCP now Disabled

;CAN Module Switch Settings
;--------------------------

;Baudrate
;8 on  7 on  Par 10-01
;8 on  7 off 500kbps
;8 off 7 on  250kbps
;8 off 7 off 125kbps

;Node Number Binary
;1 = 1s
;2 = 2s
;3 = 4s
;4 = 8s
;5 = 16s
;6 = 32s

;
;	!!! DO NOT CHANGE THE SEQUENCE OF THE PARAMETERS
;
; FU parameter to the Ubertragung (only parameter, which deviates from the default values)
;
; 1.5 kW Star
;
; Index, Subindex, Datatype (Bytes), Setting (DINT) ; Comments
0002,00,01,00000001	; [000] 00-02, Motor Speed 0 - RPM, 1 - Hz
0001,00,01,00000000	; [001] 00-01, Language 0 - English, 1 - German
0011,00,01,00000001	; [002] 00-11, Edit Setup 1
0190,00,01,00000002	; [003] 01-90, Motor Thermal Protection, 2 - Thermistor
0040,00,01,00000000 ; [---] 00-40, Hand On Key on LCP 0 - Disabled No Function
0381,00,04,00000020 ; [000] 03-81, QuickStop ramp time 100 - 1s
0458,00,01,00000001	; [004] 04-58, Missing motor phase function, 1 - Trip 100ms
0854,00,01,00000001	; [005] 08-54, Reversing select 1 - Bus only 3 - Bus and Terminal
0211,00,02,00000120	; [006] 02-11, Brake resistor 210 Ohm 150
0212,00,04,00001200	; [007] 02-12, Brake power limit 100 Watt 200
0213,00,01,00000002	; [008] 02-13, Brake check 2 - Alarm
1426,00,01,00000000 ; [---] 14-26, Trip delay at inverter fault 0 = Disabled
0803,00,04,00000002 ; [000] 08-03, Control Word Timeout Time 10 = 1Sec
0804,00,01,00000002	; [009] 08-04, Control Word Timeout Function 2 - Stop with auto restart
0801,00,01,00000000	; [010] 08-01, Control Site, 0 - Controlword only & Digital
0223,00,01,00000005	; [011] 02-23, Active brake delay 0,3 s
1761,00,01,00000002	; [012] 17-61, Encoder Signal Monitoring (Encoder faulty), 2 - Trip
1710,00,01,00000001	; [013] 17-10, Encoder Signal Type 1 - TTL
1711,00,02,00001024	; [014] 17-11, Encoder Resolution 1024 Pulse
0430,00,01,00000001 ; [015] 04-30, Motor Feedback Loss Function, 1 - Warning, 2* - Trip
0431,00,02,00000300 ; [016] 04-31, Motor Feedback Speed Error RPM, 0-600, 300*
0226,00,02,00005000	; [015] 02-26, Torque Ref, 50,00%
0228,00,02,00000200	; [016] 02-28, Gain Boost Factor, 2,00% 0-4% ***************************
0519,00,01,00000003	; [017] 05-19, Terminal 37 Safe Stop, 3 - Safe Stop Warning
0120,00,04,00000150	; [018] 01-20, Motor Power 1.5kW
0101,00,01,00000003	; [019] 01-01, Motor Control Principle, 3 - Flux with motor feedback
0122,00,02,00000400	; [020] 01-22, Motor voltage 400 V
0123,00,02,00000050	; [021] 01-23, Motor frequency 50 Hz
0162,00,02,00000100	; [022] 01-62, Slip compenstation 100%
0410,00,01,00000002	; [023] 04-10, Motor speed direction, 2 - both directions
0540,00,01,00000032	; [024] 05-40, [0] Relay 1 Function, 32 - Mech brake ctrl
0540,01,01,00000032	; [025] 05-40, [1] Relay 2 Function, 32 - Mech brake ctrl
0802,00,01,00000003 ; [---] 08-02, Control Site 3 - Option A CAN Bus
0102,00,01,00000002	; [026] 01-02, Flux Motor Feeback Source 2 - MCB102
0125,00,02,00001420	; [027] 01-25, Motor nominal speed 1420 rpm
0702,00,02,00000070	; [028] 07-02, Speed PID proportionl gain 0,070
0700,00,01,00000002	; [029] 07-00, Speed PID Feedback Source 2 - MCB102
0172,00,01,00000006	; [030] 01-72, Start function, 6 - Hoist Mech. Brake Rel
0210,00,01,00000001	; [031] 02-10, Brake Function, 1 - Resistor brake
1410,00,01,00000005	; [032] 14-10, Mains failure, 3 - Coasting 5 - Kenetic backup , trip
0193,00,01,00000006	; [033] 01-93, Thermistor source, 6 - Digital Input 33
0100,00,01,00000001	; [034] 01-00, Configuration mode, 1 - Closed loop with encoder
0139,00,01,00000004	; [035] 01-39, Motor poles, 4
0511,00,01,00000000	; [036] 05-11, Terminal 19, 0 - No Operation
0512,00,01,00000000	; [037] 05-12, Terminal 27, 0 - No Operation
0513,00,01,00000000	; [038] 05-13, Terminal 29, 0 - No Operation
0514,00,01,00000004	; [038] 05-14, Terminal 32, 4 - Quick stop
0510,00,01,00000000	; [039] 05-10, Terminal 18, 0 - No Operation
0175,00,02,00000015	; [040] 01-75, Start Speed, 1,5 Hz
0222,00,02,00000005	; [041] 02-22, Activate Brake Speed ?en bei 0,5 Hz
0124,00,04,00000360	; [042] 01-24, Motor current 5,2 A
0341,00,04,00000100	; [043] 03-41, Ramp 1 ramp up time (1 Sec to 50 Hz)
0342,00,04,00000100	; [044] 03-42, Ramp 1 ramp down time (1 Sec to  0 Hz)
0414,00,02,00001000	; [045] 04-14, Motor Speed High Limit 100,0 Hz
0220,00,04,00000180	; [046] 02-20, Release brake current 1,8 A - About Half of motor A?
;0130,00,04,00029763	; [047] 01-30, Stator resistance (Rs) 2,9763 Ohm
;0131,00,04,00022212	; [048] 01-31, Rotor resistance (Rr) 2,2212 Ohm
;0134,00,04,00031036	; [049] 01-34, Rotor leakage reactance (X2) 3,1036 Ohm
;0136,00,04,01803904	; [050] 01-36, Iron loss resistance (Rfe) 1803,904 Ohm
;0135,00,04,00653996	; [051] 01-35, Main reactance (Xh) 65,3996 Ohm
0416,00,02,00002500	; [052] 04-16, Torque limit motor mode, 160,0 - % NOW 250%
0417,00,02,00001600	; [053] 04-17, Torque limit generator mode, 160,0 %
;0133,00,04,00031036	; [054] 01-33, Stator leakage reactance (X1), 3,1036 Ohm
0303,00,04,00100000	; [055] 03-03, Maximum Reference, 100,000
0418,00,04,00001720	; [056] 04-18, Current Limit 172,0 % - NOW 250%
0851,00,01,00000003	; [0] 08-51, Quick stop Logical OR
```

### Program Logical/Robo_Drive_Control/Lift_PosMonitor (IEC) - *1ms Task to monitor and auto reference VC Works with liftv7

#### Variables.var
```iecst
VAR
	AutoRefTolerance : UINT;
	n : UINT;
	i_refSwitch : BOOL;
	refPLS : ARRAY[0..MaxRobo] OF R_TRIG;
	PositionError : DINT;
	debugRB : UINT;
	lastPosError : DINT;
END_VAR
```

#### Main.st
```iecst
PROGRAM _CYCLIC
	AutoRefTolerance := 50; //10 = 1mm
	FOR n:= 1 TO MaxRobo DO
		i_refSwitch := X[30 + (n * 2)].X04;
		refPLS[n].CLK := i_refSwitch;
		refPLS[n]();
		PositionError := 0;
		IF (RB[n].Lift.SeqStep = 30) AND refPLS[n].Q THEN
			IF RB[n].Lift.RunReverse THEN
				PositionError := (RB_Posn[n].Lift.RefOffset - RB[n].Lift.PosnNow);
				IF n = debugRB THEN
					lastPosError := PositionError;
				END_IF;
			END_IF;
			IF 	(RB[n].Lift.PosnAct > RB_Retain[n].Lift.PosnRef + AutoRefTolerance)
				OR (RB[n].Lift.PosnAct < (RB_Retain[n].Lift.PosnRef + AutoRefTolerance)) THEN//Check Hoist is going down FOR direction onto Prox
				//;MASK out +/- with ABS
				IF (ABS(PositionError) > AutoRefTolerance) THEN
					RB[n].Lift.SeqStep := 23;
				END_IF;
			END_IF;
		END_IF;
	END_FOR;

END_PROGRAM
```

### Program Logical/Robo_Drive_Control/31_vc1 (IEC)

#### vc.var
```iecst
VAR CONSTANT
	POS_FULL_BAG_OUT : USINT := 1;
	POS_FULL_BAG_IN : USINT := 4;
	POS_EMPTY_BAG_OUT : USINT := 3;
	POS_EMPTY_BAG_IN : USINT := 2;
END_VAR
VAR
	Aligned : BOOL;
	Alternator : UINT;
	AreaChoice : UINT;
	AreaEndLine : UINT := 0;
	AreaProg : UINT;
	AreaStartLine : UINT;
	AreaValid : BOOL := FALSE;
	AutoCycleET : TIME;
	AutoCycleT : BOOL;
	AutoTunePosition : UINT := 0;
	AutoTuneSequence : UINT := 0;
	CycleCount : UINT;
	DisableDrive : BOOL;
	DriveDisabled : BOOL;
	DrivePosnOk : BOOL;
	DrivesReady : BOOL;
	I_BagArriveCarr : BOOL;
	I_BagOnCarr : BOOL;
	I_LoadingMode : BOOL;
	I_PowerSave : BOOL;
	I_SafeStopOK : BOOL;
	I_UnloadingMode : BOOL;
	I_UpPushButton : BOOL;
END_VAR
VAR RETAIN
	LASTSTEP : UINT;
END_VAR
VAR
	LiftIn : FC302_ControlIn := (0);
	LiftOut : FC302_ControlOut := (0);
	myMaxWeight : ARRAY[0..4] OF UINT;
	mySeq : UINT;
	myVC : USINT;
	n : UINT;
	NoLift : BOOL;
	O_OpenCarrStop : BOOL;
	OpenStopEnabled : BOOL;
	PLS : BOOL;
	PositionSetup : BOOL;
	Posn : UINT;
	PosnOk : BOOL;
	RailAlignPosn : ARRAY[0..9] OF USINT;
	RailOkReceive : BOOL;
	RailOkRelease : BOOL;
	RequiredZone2 : BOOL;
	RequiredZone2ET : TIME;
	RotateIm : BOOL;
	RotateIn : FC302_ControlIn;
	RotateOut : FC302_ControlOut;
	Run : BOOL;
	RunMotor : BOOL;
	RunPosition : UINT;
	Status : UINT;
	STEP : UINT;
	TimerAlarm : TON_10ms;
	ValidCat : BOOL;
	ValidCus : BOOL;
	ValidDst : BOOL;
	ValidPrg : BOOL;
	ValidWgt : BOOL;
	VCAction : UINT;
	VCActionDisabled : BOOL;
	VCActionDisabledET : TIME := T#0ms;
	VCHeartBeat : UINT;
	VCIndex : UINT;
	VCInit : BOOL;
	VCMode : UINT;
	myBag : UINT;
	myDisplayBag : UINT;
	myRelLine : UINT;
	I_BagAtOutbuffer : BOOL;
	I_OutbufferOpen : BOOL;
	DataValid : BOOL;
	Dest : UINT;
	myZone : UINT;
	myIO : UINT;
	GetFullBag : BOOL;
	GetEmpty : BOOL;
	myBufferBag : UINT;
	almDisableSequence : BOOL;
	SettledCarriage : BOOL;
	SettledCarriageET : UDINT;
	CarriageClear : BOOL;
	CarriageClearET : UDINT;
	EmptySpace : UINT;
	SPNBufferSpace : UINT;
	BothVCGetFullBag : BOOL;
	OtherVCisGettingEmpty : BOOL;
	BufferStopOpen : ARRAY[0..49] OF BOOL;
	BagAtBuffer : ARRAY[0..49] OF BOOL;
	LineValid : ARRAY[0..9] OF BOOL;
	WaitTime : ARRAY[0..9] OF UDINT;
	WaitingLongest : UINT;
	O_OpenIngoingStop : BOOL;
	O_OpenBuffer : BOOL;
	O_Lamp : BOOL;
	O_SafeStopEmptyIn : BOOL;
	DataEntryBag : UINT;
	BuffOutClear : BOOL;
	BulkMode : BOOL;
	GetBag : ARRAY[0..8] OF BOOL;
	PButton : BOOL;
	PButtonET : UDINT;
	CartInVC : BOOL;
	LineOffset : BOOL;
	I_BagReleased : BOOL;
	myFullRelLine : UINT;
	myFullRelBag : UINT;
	HaltSysZoneClear : BOOL;
	HaltSysZoneClearET : TIME;
	SettledCarriage12 : BOOL;
	SettledCarriage12ET : TIME;
	stopZone : BOOL;
	myEmptyRelLine : UINT;
	myEmptyRelBag : UINT;
	releaseValid : BOOL;
	myFullBuffBag : UINT;
	I_BagAtFullBuffer : BOOL;
	SettledFullBuffer : BOOL;
	SettledFullBufferET : UDINT;
	myFullLine : USINT;
	O_OpenFullBagBuffer : BOOL;
	raw : DINT;
	myWeighBag : UINT;
	myHttp : UINT;
	requestURL : STRING[100];
	requestData : STRING[256];
	batchString : STRING[15];
	weightString : STRING[15];
	httpComplete : BOOL;
	myReportStn : UINT;
	weightOk : BOOL;
	weightOkET : UDINT;
END_VAR
```
